LIN {X 0,Y 136.364,Z 311.031,A -85,B 0,C 180,E1 -25968.178,E2 -25968.178} C_VEL
LIN {X 0,Y 134.01,Z 323.173,A -85,B 0,C 180,E1 -25969.777,E2 -25969.777} C_VEL
LIN {X 0,Y 130.975,Z 334.933,A -85,B 0,C 180,E1 -25971.894,E2 -25971.894} C_VEL
LIN {X 0,Y 127.616,Z 346.371,A -85,B 0,C 180,E1 -25974.669,E2 -25974.669} C_VEL
LIN {X 0,Y 124.044,Z 357.11,A -85,B 0,C 180,E1 -25978.099,E2 -25978.099} C_VEL
LIN {X 0,Y 121.088,Z 365.283,A -85,B 0,C 180,E1 -25981.449,E2 -25981.449} C_VEL
LIN {X 0,Y 117.764,Z 374.351,A -85,B 0,C 180,E1 -25986.241,E2 -25986.241} C_VEL
LIN {X 0,Y 115.11,Z 381.715,A -85,B 0,C 180,E1 -25991.301,E2 -25991.301} C_VEL
LIN {X 0,Y 113.643,Z 386.688,A -85,B 0,C 180,E1 -25995.674,E2 -25995.674} C_VEL
LIN {X 0,Y 112.563,Z 391.484,A -85,B 0,C 180,E1 -26001.016,E2 -26001.016} C_VEL
LIN {X 0,Y 112.161,Z 395.114,A -85,B 0,C 180,E1 -26006.404,E2 -26006.404} C_VEL
LIN {X 0,Y 112.247,Z 396.97,A -85,B 0,C 180,E1 -26009.996,E2 -26009.996} C_VEL
LIN {X 0,Y 112.19,Z 398.332,A -85,B 0,C 180,E1 -26013.588,E2 -26013.588} C_VEL
LIN {X 0,Y 112.424,Z 399.289,A -85,B 0,C 180,E1 -26017.178,E2 -26017.178} C_VEL
LIN {X 0,Y 113.828,Z 400.074,A -85,B 0,C 180,E1 -26024.294,E2 -26024.294} C_VEL
LIN {X 0,Y 115.126,Z 399.897,A -85,B 0,C 180,E1 -26027.768,E2 -26027.768} C_VEL
LIN {X 0,Y 118.896,Z 398.375,A -85,B 0,C 180,E1 -26034.438,E2 -26034.438} C_VEL
LIN {X 0,Y 124.439,Z 395.336,A -85,B 0,C 180,E1 -26040.546,E2 -26040.546} C_VEL
LIN {X 0,Y 129.4,Z 391.954,A -85,B 0,C 180,E1 -26044.765,E2 -26044.765} C_VEL
LIN {X 0,Y 134.835,Z 387.585,A -85,B 0,C 180,E1 -26048.712,E2 -26048.712} C_VEL
LIN {X 0,Y 142.27,Z 381.015,A -85,B 0,C 180,E1 -26052.779,E2 -26052.779} C_VEL
LIN {X 0,Y 149.064,Z 373.931,A -85,B 0,C 180,E1 -26055.967,E2 -26055.967} C_VEL
LIN {X 0,Y 156.427,Z 365.2,A -85,B 0,C 180,E1 -26058.806,E2 -26058.806} C_VEL
LIN {X 0,Y 159.478,Z 361.16,A -85,B 0,C 180,E1 -26059.858,E2 -26059.858} C_VEL
LIN {X 0,Y 162.144,Z 357.028,A -85,B 0,C 180,E1 -26061.026,E2 -26061.026} C_VEL
LIN {X 0,Y 165.372,Z 350.19,A -85,B 0,C 180,E1 -26063.269,E2 -26063.269} C_VEL
LIN {X 0,Y 168.431,Z 342.958,A -85,B 0,C 180,E1 -26065.313,E2 -26065.313} C_VEL
LIN {X 0,Y 170.733,Z 338.125,A -85,B 0,C 180,E1 -26066.161,E2 -26066.161} C_VEL
LIN {X 0,Y 176.097,Z 326.328,A -85,B 0,C 180,E1 -26067.398,E2 -26067.398} C_VEL
LIN {X 0,Y 180.609,Z 313.511,A -85,B 0,C 180,E1 -26068.352,E2 -26068.352} C_VEL
LIN {X 0,Y 183.995,Z 300.204,A -85,B 0,C 180,E1 -26069.022,E2 -26069.022} C_VEL
LIN {X 0,Y 186.074,Z 287.077,A -85,B 0,C 180,E1 -26069.451,E2 -26069.451} C_VEL
LIN {X 0,Y 186.09,Z 286.042,A -85,B 0,C 180,E1 -26069.608,E2 -26069.608} C_VEL
LIN {X 0,Y 184.683,Z 281.104,A -85,B 0,C 180,E1 -26072.259,E2 -26072.259} C_VEL
LIN {X 0,Y 183.758,Z 278.277,A -85,B 0,C 180,E1 -26074.485,E2 -26074.485} C_VEL
LIN {X 0,Y 183.075,Z 275.937,A -85,B 0,C 180,E1 -26076.697,E2 -26076.697} C_VEL
LIN {X 0,Y 182.587,Z 274.798,A -85,B 0,C 180,E1 -26078.942,E2 -26078.942} C_VEL
LIN {X 0,Y 182.267,Z 274.378,A -85,B 0,C 180,E1 -26082.032,E2 -26082.032} C_VEL
LIN {X 0,Y 182.898,Z 274.923,A -85,B 0,C 180,E1 -26086.669,E2 -26086.669} C_VEL
LIN {X 0,Y 183.255,Z 275.583,A -85,B 0,C 180,E1 -26087.91,E2 -26087.91} C_VEL
LIN {X 0,Y 184.929,Z 279.204,A -85,B 0,C 180,E1 -26091.984,E2 -26091.984} C_VEL
LIN {X 0,Y 186.439,Z 283.928,A -85,B 0,C 180,E1 -26094.713,E2 -26094.713} C_VEL
LIN {X 0,Y 184.015,Z 299.42,A -85,B 0,C 180,E1 -26095.227,E2 -26095.227} C_VEL
LIN {X 0,Y 180.609,Z 312.589,A -85,B 0,C 180,E1 -26095.931,E2 -26095.931} C_VEL
LIN {X 0,Y 176.382,Z 324.717,A -85,B 0,C 180,E1 -26096.929,E2 -26096.929} C_VEL
LIN {X 0,Y 171.678,Z 335.275,A -85,B 0,C 180,E1 -26098.074,E2 -26098.074} C_VEL
LIN {X 0,Y 165.53,Z 346.46,A -85,B 0,C 180,E1 -26099.672,E2 -26099.672} C_VEL
LIN {X 0,Y 158.442,Z 357.17,A -85,B 0,C 180,E1 -26101.789,E2 -26101.789} C_VEL
LIN {X 0,Y 151.478,Z 365.954,A -85,B 0,C 180,E1 -26104.089,E2 -26104.089} C_VEL
LIN {X 0,Y 145.01,Z 372.979,A -85,B 0,C 180,E1 -26106.549,E2 -26106.549} C_VEL
LIN {X 0,Y 137.992,Z 379.587,A -85,B 0,C 180,E1 -26109.65,E2 -26109.65} C_VEL
LIN {X 0,Y 130.279,Z 385.85,A -85,B 0,C 180,E1 -26113.845,E2 -26113.845} C_VEL
LIN {X 0,Y 122.865,Z 390.935,A -85,B 0,C 180,E1 -26118.918,E2 -26118.918} C_VEL
LIN {X 0,Y 116.03,Z 394.604,A -85,B 0,C 180,E1 -26125.085,E2 -26125.085} C_VEL
LIN {X 0,Y 111.896,Z 396.254,A -85,B 0,C 180,E1 -26130.162,E2 -26130.162} C_VEL
LIN {X 0,Y 108.662,Z 396.997,A -85,B 0,C 180,E1 -26135.596,E2 -26135.596} C_VEL
LIN {X 0,Y 105.831,Z 396.588,A -85,B 0,C 180,E1 -26143.08,E2 -26143.08} C_VEL
LIN {X 0,Y 104.833,Z 395.519,A -85,B 0,C 180,E1 -26147.909,E2 -26147.909} C_VEL
LIN {X 0,Y 104.419,Z 393.352,A -85,B 0,C 180,E1 -26153.866,E2 -26153.866} C_VEL
LIN {X 0,Y 104.975,Z 389.721,A -85,B 0,C 180,E1 -26160.494,E2 -26160.494} C_VEL
LIN {X 0,Y 106.235,Z 385.043,A -85,B 0,C 180,E1 -26166.618,E2 -26166.618} C_VEL
LIN {X 0,Y 108.263,Z 378.481,A -85,B 0,C 180,E1 -26173.021,E2 -26173.021} C_VEL
LIN {X 0,Y 110.851,Z 371.57,A -85,B 0,C 180,E1 -26178.113,E2 -26178.113} C_VEL
LIN {X 0,Y 114.059,Z 363.129,A -85,B 0,C 180,E1 -26182.925,E2 -26182.925} C_VEL
LIN {X 0,Y 117.876,Z 353.263,A -85,B 0,C 180,E1 -26187.218,E2 -26187.218} C_VEL
LIN {X 0,Y 121.724,Z 342.211,A -85,B 0,C 180,E1 -26190.831,E2 -26190.831} C_VEL
LIN {X 0,Y 125.277,Z 330.465,A -85,B 0,C 180,E1 -26193.735,E2 -26193.735} C_VEL
LIN {X 0,Y 128.149,Z 319.202,A -85,B 0,C 180,E1 -26195.808,E2 -26195.808} C_VEL
LIN {X 0,Y 130.747,Z 305.847,A -85,B 0,C 180,E1 -26197.58,E2 -26197.58} C_VEL
LIN {X 0,Y 132.648,Z 292.684,A -85,B 0,C 180,E1 -26198.717,E2 -26198.717} C_VEL
LIN {X 0,Y 136.222,Z 248.968,A -85,B 0,C 180,E1 -26200.99,E2 -26200.99} C_VEL
LIN {X 0,Y 132.344,Z 237.4,A -85,B 0,C 180,E1 -26203.135,E2 -26203.135} C_VEL
LIN {X 0,Y 124.67,Z 222.791,A -85,B 0,C 180,E1 -26207.139,E2 -26207.139} C_VEL
LIN {X 0,Y 118.536,Z 212.859,A -85,B 0,C 180,E1 -26210.752,E2 -26210.752} C_VEL
LIN {X 0,Y 115.586,Z 208.527,A -85,B 0,C 180,E1 -26212.616,E2 -26212.616} C_VEL
LIN {X 0,Y 113.611,Z 205.554,A -85,B 0,C 180,E1 -26213.954,E2 -26213.954} C_VEL
LIN {X 0,Y 111.26,Z 202.05,A -85,B 0,C 180,E1 -26215.65,E2 -26215.65} C_VEL
LIN {X 0,Y 108.737,Z 199.33,A -85,B 0,C 180,E1 -26217.499,E2 -26217.499} C_VEL
LIN {X 0,Y 107.886,Z 197.158,A -85,B 0,C 180,E1 -26218.585,E2 -26218.585} C_VEL
LIN {X 0,Y 107.828,Z 196.58,A -85,B 0,C 180,E1 -26219.804,E2 -26219.804} C_VEL
LIN {X 0,Y 107.715,Z 196.516,A -85,B 0,C 180,E1 -26225.964,E2 -26225.964} C_VEL
LIN {X 0,Y 107.685,Z 196.561,A -85,B 0,C 180,E1 -26230.746,E2 -26230.746} C_VEL
LIN {X 0,Y 107.677,Z 196.518,A -85,B 0,C 180,E1 -26235.891,E2 -26235.891} C_VEL
LIN {X 0,Y 107.687,Z 196.523,A -85,B 0,C 180,E1 -26241.556,E2 -26241.556} C_VEL
LIN {X 0,Y 107.794,Z 196.539,A -85,B 0,C 180,E1 -26248.563,E2 -26248.563} C_VEL
LIN {X 0,Y 107.914,Z 196.522,A -85,B 0,C 180,E1 -26257,E2 -26257} C_VEL
LIN {X 0,Y 108.034,Z 196.506,A -85,B 0,C 180,E1 -26264.919,E2 -26264.919} C_VEL
LIN {X 0,Y 108.254,Z 196.498,A -85,B 0,C 180,E1 -26268.771,E2 -26268.771} C_VEL
LIN {X 0,Y 108.417,Z 196.48,A -85,B 0,C 180,E1 -26276.285,E2 -26276.285} C_VEL
LIN {X 0,Y 108.882,Z 196.374,A -85,B 0,C 180,E1 -26280.002,E2 -26280.002} C_VEL
LIN {X 0,Y 108.295,Z 196.461,A -85,B 0,C 180,E1 -26287.459,E2 -26287.459} C_VEL
LIN {X 0,Y 108.144,Z 196.479,A -85,B 0,C 180,E1 -26292.874,E2 -26292.874} C_VEL
LIN {X 0,Y 107.867,Z 196.515,A -85,B 0,C 180,E1 -26299.014,E2 -26299.014} C_VEL
LIN {X 0,Y 107.826,Z 196.672,A -85,B 0,C 180,E1 -26304.492,E2 -26304.492} C_VEL
LIN {X 0,Y 107.991,Z 197.518,A -85,B 0,C 180,E1 -26305.45,E2 -26305.45} C_VEL
LIN {X 0,Y 109.583,Z 200.432,A -85,B 0,C 180,E1 -26306.935,E2 -26306.935} C_VEL
LIN {X 0,Y 111.163,Z 201.973,A -85,B 0,C 180,E1 -26308.052,E2 -26308.052} C_VEL
LIN {X 0,Y 113.296,Z 205.383,A -85,B 0,C 180,E1 -26309.616,E2 -26309.616} C_VEL
LIN {X 0,Y 114.635,Z 207.06,A -85,B 0,C 180,E1 -26310.503,E2 -26310.503} C_VEL
LIN {X 0,Y 119.745,Z 215.159,A -85,B 0,C 180,E1 -26313.818,E2 -26313.818} C_VEL
LIN {X 0,Y 125.181,Z 224.549,A -85,B 0,C 180,E1 -26316.989,E2 -26316.989} C_VEL
LIN {X 0,Y 128.209,Z 230.807,A -85,B 0,C 180,E1 -26318.671,E2 -26318.671} C_VEL
LIN {X 0,Y 133.626,Z 245.521,A -85,B 0,C 180,E1 -26321.702,E2 -26321.702} C_VEL
LIN {X 0,Y 136.062,Z 253.151,A -85,B 0,C 180,E1 -26323.047,E2 -26323.047} C_VEL
LIN {X 0,Y 132.47,Z 297.001,A -85,B 0,C 180,E1 -26325.357,E2 -26325.357} C_VEL
LIN {X 0,Y 130.339,Z 310.747,A -85,B 0,C 180,E1 -26326.564,E2 -26326.564} C_VEL
LIN {X 0,Y 127.891,Z 322.942,A -85,B 0,C 180,E1 -26328.214,E2 -26328.214} C_VEL
LIN {X 0,Y 124.498,Z 335.522,A -85,B 0,C 180,E1 -26330.571,E2 -26330.571} C_VEL
LIN {X 0,Y 120.993,Z 346.834,A -85,B 0,C 180,E1 -26333.457,E2 -26333.457} C_VEL
LIN {X 0,Y 117.286,Z 357.395,A -85,B 0,C 180,E1 -26337.028,E2 -26337.028} C_VEL
LIN {X 0,Y 114.255,Z 365.435,A -85,B 0,C 180,E1 -26340.518,E2 -26340.518} C_VEL
LIN {X 0,Y 110.755,Z 374.55,A -85,B 0,C 180,E1 -26345.637,E2 -26345.637} C_VEL
LIN {X 0,Y 107.985,Z 381.855,A -85,B 0,C 180,E1 -26351.006,E2 -26351.006} C_VEL
LIN {X 0,Y 106.273,Z 387.67,A -85,B 0,C 180,E1 -26356.613,E2 -26356.613} C_VEL
LIN {X 0,Y 105.316,Z 392.2,A -85,B 0,C 180,E1 -26362.326,E2 -26362.326} C_VEL
LIN {X 0,Y 105.089,Z 394.568,A -85,B 0,C 180,E1 -26366.161,E2 -26366.161} C_VEL
LIN {X 0,Y 105.169,Z 396.493,A -85,B 0,C 180,E1 -26369.996,E2 -26369.996} C_VEL
LIN {X 0,Y 105.108,Z 397.968,A -85,B 0,C 180,E1 -26373.83,E2 -26373.83} C_VEL
LIN {X 0,Y 105.368,Z 399.005,A -85,B 0,C 180,E1 -26377.662,E2 -26377.662} C_VEL
LIN {X 0,Y 106.944,Z 399.927,A -85,B 0,C 180,E1 -26385.236,E2 -26385.236} C_VEL
LIN {X 0,Y 110.154,Z 399.374,A -85,B 0,C 180,E1 -26392.503,E2 -26392.503} C_VEL
LIN {X 0,Y 115.22,Z 397.265,A -85,B 0,C 180,E1 -26399.202,E2 -26399.202} C_VEL
LIN {X 0,Y 121.822,Z 393.613,A -85,B 0,C 180,E1 -26405.228,E2 -26405.228} C_VEL
LIN {X 0,Y 127.627,Z 389.555,A -85,B 0,C 180,E1 -26409.56,E2 -26409.56} C_VEL
LIN {X 0,Y 133.755,Z 384.791,A -85,B 0,C 180,E1 -26413.079,E2 -26413.079} C_VEL
LIN {X 0,Y 141.886,Z 377.496,A -85,B 0,C 180,E1 -26416.932,E2 -26416.932} C_VEL
LIN {X 0,Y 148.117,Z 371.086,A -85,B 0,C 180,E1 -26419.387,E2 -26419.387} C_VEL
LIN {X 0,Y 155.894,Z 361.713,A -85,B 0,C 180,E1 -26422.081,E2 -26422.081} C_VEL
LIN {X 0,Y 163.321,Z 351.079,A -85,B 0,C 180,E1 -26424.308,E2 -26424.308} C_VEL
LIN {X 0,Y 169.699,Z 340.099,A -85,B 0,C 180,E1 -26425.918,E2 -26425.918} C_VEL
LIN {X 0,Y 170.733,Z 338.125,A -85,B 0,C 180,E1 -26426.161,E2 -26426.161} C_VEL
LIN {X 0,Y 172.97,Z 333.179,A -85,B 0,C 180,E1 -26426.963,E2 -26426.963} C_VEL
LIN {X 0,Y 175.622,Z 325.109,A -85,B 0,C 180,E1 -26428.674,E2 -26428.674} C_VEL
LIN {X 0,Y 177.866,Z 316.694,A -85,B 0,C 180,E1 -26430.186,E2 -26430.186} C_VEL
LIN {X 0,Y 179.367,Z 311.228,A -85,B 0,C 180,E1 -26430.68,E2 -26430.68} C_VEL
LIN {X 0,Y 182.606,Z 297.924,A -85,B 0,C 180,E1 -26431.236,E2 -26431.236} C_VEL
LIN {X 0,Y 183.837,Z 290.196,A -85,B 0,C 180,E1 -26431.549,E2 -26431.549} C_VEL
LIN {X 0,Y 182.832,Z 286.166,A -85,B 0,C 180,E1 -26434.026,E2 -26434.026} C_VEL
LIN {X 0,Y 181.855,Z 282.714,A -85,B 0,C 180,E1 -26437.264,E2 -26437.264} C_VEL
LIN {X 0,Y 181.445,Z 281.701,A -85,B 0,C 180,E1 -26439.597,E2 -26439.597} C_VEL
LIN {X 0,Y 181.41,Z 281.461,A -85,B 0,C 180,E1 -26444.264,E2 -26444.264} C_VEL
LIN {X 0,Y 182.006,Z 282.25,A -85,B 0,C 180,E1 -26447.261,E2 -26447.261} C_VEL
LIN {X 0,Y 183.546,Z 285.951,A -85,B 0,C 180,E1 -26451.418,E2 -26451.418} C_VEL
LIN {X 0,Y 184.109,Z 288.316,A -85,B 0,C 180,E1 -26452.72,E2 -26452.72} C_VEL
LIN {X 0,Y 181.696,Z 301.571,A -85,B 0,C 180,E1 -26453.168,E2 -26453.168} C_VEL
LIN {X 0,Y 178.406,Z 313.577,A -85,B 0,C 180,E1 -26453.804,E2 -26453.804} C_VEL
LIN {X 0,Y 173.621,Z 326.545,A -85,B 0,C 180,E1 -26454.856,E2 -26454.856} C_VEL
LIN {X 0,Y 168.174,Z 337.859,A -85,B 0,C 180,E1 -26456.089,E2 -26456.089} C_VEL
LIN {X 0,Y 161.769,Z 348.678,A -85,B 0,C 180,E1 -26457.663,E2 -26457.663} C_VEL
LIN {X 0,Y 154.609,Z 358.712,A -85,B 0,C 180,E1 -26459.664,E2 -26459.664} C_VEL
LIN {X 0,Y 147.654,Z 366.91,A -85,B 0,C 180,E1 -26461.829,E2 -26461.829} C_VEL
LIN {X 0,Y 139.77,Z 374.876,A -85,B 0,C 180,E1 -26464.696,E2 -26464.696} C_VEL
LIN {X 0,Y 131.62,Z 381.86,A -85,B 0,C 180,E1 -26468.216,E2 -26468.216} C_VEL
LIN {X 0,Y 125.487,Z 386.383,A -85,B 0,C 180,E1 -26471.47,E2 -26471.47} C_VEL
LIN {X 0,Y 117.415,Z 391.414,A -85,B 0,C 180,E1 -26476.74,E2 -26476.74} C_VEL
LIN {X 0,Y 110.769,Z 394.663,A -85,B 0,C 180,E1 -26482.374,E2 -26482.374} C_VEL
LIN {X 0,Y 104.866,Z 396.715,A -85,B 0,C 180,E1 -26489.406,E2 -26489.406} C_VEL
LIN {X 0,Y 101.996,Z 397.143,A -85,B 0,C 180,E1 -26494.232,E2 -26494.232} C_VEL
LIN {X 0,Y 99.83,Z 396.974,A -85,B 0,C 180,E1 -26499.314,E2 -26499.314} C_VEL
LIN {X 0,Y 98.047,Z 395.858,A -85,B 0,C 180,E1 -26505.788,E2 -26505.788} C_VEL
LIN {X 0,Y 97.334,Z 393.636,A -85,B 0,C 180,E1 -26512.582,E2 -26512.582} C_VEL
LIN {X 0,Y 97.743,Z 390.021,A -85,B 0,C 180,E1 -26519.786,E2 -26519.786} C_VEL
LIN {X 0,Y 98.644,Z 386.73,A -85,B 0,C 180,E1 -26524.698,E2 -26524.698} C_VEL
LIN {X 0,Y 100.166,Z 381.698,A -85,B 0,C 180,E1 -26530.537,E2 -26530.537} C_VEL
LIN {X 0,Y 102.434,Z 375.417,A -85,B 0,C 180,E1 -26536.176,E2 -26536.176} C_VEL
LIN {X 0,Y 105.445,Z 367.905,A -85,B 0,C 180,E1 -26541.379,E2 -26541.379} C_VEL
LIN {X 0,Y 109.234,Z 358.584,A -85,B 0,C 180,E1 -26546.315,E2 -26546.315} C_VEL
LIN {X 0,Y 113.17,Z 348.266,A -85,B 0,C 180,E1 -26550.448,E2 -26550.448} C_VEL
LIN {X 0,Y 117.139,Z 336.881,A -85,B 0,C 180,E1 -26553.832,E2 -26553.832} C_VEL
LIN {X 0,Y 120.48,Z 325.56,A -85,B 0,C 180,E1 -26556.374,E2 -26556.374} C_VEL
LIN {X 0,Y 123.345,Z 313.358,A -85,B 0,C 180,E1 -26558.399,E2 -26558.399} C_VEL
LIN {X 0,Y 125.893,Z 299.378,A -85,B 0,C 180,E1 -26559.963,E2 -26559.963} C_VEL
LIN {X 0,Y 127.481,Z 285.745,A -85,B 0,C 180,E1 -26560.887,E2 -26560.887} C_VEL
LIN {X 0,Y 130.367,Z 250.585,A -85,B 0,C 180,E1 -26562.745,E2 -26562.745} C_VEL
LIN {X 0,Y 127.215,Z 241.064,A -85,B 0,C 180,E1 -26564.606,E2 -26564.606} C_VEL
LIN {X 0,Y 120.126,Z 227.179,A -85,B 0,C 180,E1 -26568.658,E2 -26568.658} C_VEL
LIN {X 0,Y 112.976,Z 215.35,A -85,B 0,C 180,E1 -26573.258,E2 -26573.258} C_VEL
LIN {X 0,Y 107.405,Z 207.315,A -85,B 0,C 180,E1 -26577.398,E2 -26577.398} C_VEL
LIN {X 0,Y 105.019,Z 204.269,A -85,B 0,C 180,E1 -26579.38,E2 -26579.38} C_VEL
LIN {X 0,Y 104.123,Z 202.586,A -85,B 0,C 180,E1 -26580.229,E2 -26580.229} C_VEL
LIN {X 0,Y 101.914,Z 200.528,A -85,B 0,C 180,E1 -26582.126,E2 -26582.126} C_VEL
LIN {X 0,Y 100.774,Z 198.106,A -85,B 0,C 180,E1 -26583.646,E2 -26583.646} C_VEL
LIN {X 0,Y 100.667,Z 197.442,A -85,B 0,C 180,E1 -26585.172,E2 -26585.172} C_VEL
LIN {X 0,Y 100.643,Z 197.42,A -85,B 0,C 180,E1 -26589.816,E2 -26589.816} C_VEL
LIN {X 0,Y 100.648,Z 197.392,A -85,B 0,C 180,E1 -26595.714,E2 -26595.714} C_VEL
LIN {X 0,Y 100.625,Z 197.394,A -85,B 0,C 180,E1 -26601.056,E2 -26601.056} C_VEL
LIN {X 0,Y 100.691,Z 197.432,A -85,B 0,C 180,E1 -26606.891,E2 -26606.891} C_VEL
LIN {X 0,Y 100.791,Z 197.413,A -85,B 0,C 180,E1 -26615.27,E2 -26615.27} C_VEL
LIN {X 0,Y 100.819,Z 197.419,A -85,B 0,C 180,E1 -26619.604,E2 -26619.604} C_VEL
LIN {X 0,Y 101.104,Z 197.376,A -85,B 0,C 180,E1 -26626.713,E2 -26626.713} C_VEL
LIN {X 0,Y 101.236,Z 197.354,A -85,B 0,C 180,E1 -26632.021,E2 -26632.021} C_VEL
LIN {X 0,Y 101.814,Z 197.251,A -85,B 0,C 180,E1 -26640.002,E2 -26640.002} C_VEL
LIN {X 0,Y 101.232,Z 197.345,A -85,B 0,C 180,E1 -26647.983,E2 -26647.983} C_VEL
LIN {X 0,Y 101.057,Z 197.355,A -85,B 0,C 180,E1 -26653.172,E2 -26653.172} C_VEL
LIN {X 0,Y 100.846,Z 197.647,A -85,B 0,C 180,E1 -26659.598,E2 -26659.598} C_VEL
LIN {X 0,Y 101.057,Z 198.693,A -85,B 0,C 180,E1 -26660.616,E2 -26660.616} C_VEL
LIN {X 0,Y 102.615,Z 201.345,A -85,B 0,C 180,E1 -26662.263,E2 -26662.263} C_VEL
LIN {X 0,Y 104.417,Z 202.965,A -85,B 0,C 180,E1 -26663.82,E2 -26663.82} C_VEL
LIN {X 0,Y 106.359,Z 206.215,A -85,B 0,C 180,E1 -26665.569,E2 -26665.569} C_VEL
LIN {X 0,Y 107.854,Z 207.998,A -85,B 0,C 180,E1 -26666.747,E2 -26666.747} C_VEL
LIN {X 0,Y 110.495,Z 211.755,A -85,B 0,C 180,E1 -26668.753,E2 -26668.753} C_VEL
LIN {X 0,Y 115.819,Z 220.467,A -85,B 0,C 180,E1 -26672.475,E2 -26672.475} C_VEL
LIN {X 0,Y 120.665,Z 229.07,A -85,B 0,C 180,E1 -26675.528,E2 -26675.528} C_VEL
LIN {X 0,Y 123.53,Z 235.191,A -85,B 0,C 180,E1 -26677.266,E2 -26677.266} C_VEL
LIN {X 0,Y 128.851,Z 250.363,A -85,B 0,C 180,E1 -26680.499,E2 -26680.499} C_VEL
LIN {X 0,Y 130.228,Z 254.712,A -85,B 0,C 180,E1 -26681.305,E2 -26681.305} C_VEL
LIN {X 0,Y 126.627,Z 296.718,A -85,B 0,C 180,E1 -26683.574,E2 -26683.574} C_VEL
LIN {X 0,Y 124.551,Z 309.644,A -85,B 0,C 180,E1 -26684.711,E2 -26684.711} C_VEL
LIN {X 0,Y 122.12,Z 321.52,A -85,B 0,C 180,E1 -26686.318,E2 -26686.318} C_VEL
LIN {X 0,Y 119.059,Z 332.845,A -85,B 0,C 180,E1 -26688.384,E2 -26688.384} C_VEL
LIN {X 0,Y 115.342,Z 344.634,A -85,B 0,C 180,E1 -26691.347,E2 -26691.347} C_VEL
LIN {X 0,Y 111.507,Z 355.231,A -85,B 0,C 180,E1 -26694.888,E2 -26694.888} C_VEL
LIN {X 0,Y 108.042,Z 363.889,A -85,B 0,C 180,E1 -26698.638,E2 -26698.638} C_VEL
LIN {X 0,Y 104.836,Z 371.89,A -85,B 0,C 180,E1 -26703.091,E2 -26703.091} C_VEL
LIN {X 0,Y 101.688,Z 379.657,A -85,B 0,C 180,E1 -26708.721,E2 -26708.721} C_VEL
LIN {X 0,Y 99.373,Z 386.808,A -85,B 0,C 180,E1 -26715.664,E2 -26715.664} C_VEL
LIN {X 0,Y 98.281,Z 391.513,A -85,B 0,C 180,E1 -26721.773,E2 -26721.773} C_VEL
LIN {X 0,Y 97.986,Z 395.062,A -85,B 0,C 180,E1 -26727.941,E2 -26727.941} C_VEL
LIN {X 0,Y 98.077,Z 396.001,A -85,B 0,C 180,E1 -26729.996,E2 -26729.996} C_VEL
LIN {X 0,Y 98.049,Z 397.551,A -85,B 0,C 180,E1 -26734.106,E2 -26734.106} C_VEL
LIN {X 0,Y 98.325,Z 398.701,A -85,B 0,C 180,E1 -26738.214,E2 -26738.214} C_VEL
LIN {X 0,Y 100.1,Z 399.78,A -85,B 0,C 180,E1 -26746.306,E2 -26746.306} C_VEL
LIN {X 0,Y 103.606,Z 399.379,A -85,B 0,C 180,E1 -26754.012,E2 -26754.012} C_VEL
LIN {X 0,Y 109.089,Z 397.487,A -85,B 0,C 180,E1 -26761.019,E2 -26761.019} C_VEL
LIN {X 0,Y 116.092,Z 393.991,A -85,B 0,C 180,E1 -26767.251,E2 -26767.251} C_VEL
LIN {X 0,Y 121.863,Z 390.377,A -85,B 0,C 180,E1 -26771.431,E2 -26771.431} C_VEL
LIN {X 0,Y 128.71,Z 385.565,A -85,B 0,C 180,E1 -26775.217,E2 -26775.217} C_VEL
LIN {X 0,Y 137.192,Z 378.554,A -85,B 0,C 180,E1 -26779.073,E2 -26779.073} C_VEL
LIN {X 0,Y 144.984,Z 370.969,A -85,B 0,C 180,E1 -26781.966,E2 -26781.966} C_VEL
LIN {X 0,Y 153.104,Z 361.599,A -85,B 0,C 180,E1 -26784.56,E2 -26784.56} C_VEL
LIN {X 0,Y 160.092,Z 352.085,A -85,B 0,C 180,E1 -26786.515,E2 -26786.515} C_VEL
LIN {X 0,Y 166.667,Z 341.487,A -85,B 0,C 180,E1 -26788.057,E2 -26788.057} C_VEL
LIN {X 0,Y 172.591,Z 329.645,A -85,B 0,C 180,E1 -26789.335,E2 -26789.335} C_VEL
LIN {X 0,Y 177.488,Z 317.232,A -85,B 0,C 180,E1 -26790.297,E2 -26790.297} C_VEL
LIN {X 0,Y 179.367,Z 311.228,A -85,B 0,C 180,E1 -26790.68,E2 -26790.68} C_VEL
LIN {X 0,Y 180.694,Z 305.957,A -85,B 0,C 180,E1 -26791.095,E2 -26791.095} C_VEL
LIN {X 0,Y 181.439,Z 300.97,A -85,B 0,C 180,E1 -26791.859,E2 -26791.859} C_VEL
LIN {X 0,Y 181.708,Z 296.632,A -85,B 0,C 180,E1 -26792.923,E2 -26792.923} C_VEL
LIN {X 0,Y 181.57,Z 293.696,A -85,B 0,C 180,E1 -26794.114,E2 -26794.114} C_VEL
LIN {X 0,Y 181.523,Z 293.372,A -85,B 0,C 180,E1 -26794.303,E2 -26794.303} C_VEL
LIN {X 0,Y 180.725,Z 289.644,A -85,B 0,C 180,E1 -26797.59,E2 -26797.59} C_VEL
LIN {X 0,Y 180.365,Z 288.671,A -85,B 0,C 180,E1 -26799.929,E2 -26799.929} C_VEL
LIN {X 0,Y 180.363,Z 288.482,A -85,B 0,C 180,E1 -26804.17,E2 -26804.17} C_VEL
LIN {X 0,Y 180.84,Z 289.17,A -85,B 0,C 180,E1 -26806.846,E2 -26806.846} C_VEL
LIN {X 0,Y 182.003,Z 292.397,A -85,B 0,C 180,E1 -26810.59,E2 -26810.59} C_VEL
LIN {X 0,Y 180.306,Z 301.139,A -85,B 0,C 180,E1 -26810.954,E2 -26810.954} C_VEL
LIN {X 0,Y 176.611,Z 314.215,A -85,B 0,C 180,E1 -26811.6,E2 -26811.6} C_VEL
LIN {X 0,Y 171.863,Z 326.591,A -85,B 0,C 180,E1 -26812.559,E2 -26812.559} C_VEL
LIN {X 0,Y 166.139,Z 338.122,A -85,B 0,C 180,E1 -26813.739,E2 -26813.739} C_VEL
LIN {X 0,Y 159.814,Z 348.502,A -85,B 0,C 180,E1 -26815.162,E2 -26815.162} C_VEL
LIN {X 0,Y 152.786,Z 358.147,A -85,B 0,C 180,E1 -26816.971,E2 -26816.971} C_VEL
LIN {X 0,Y 144.672,Z 367.339,A -85,B 0,C 180,E1 -26819.266,E2 -26819.266} C_VEL
LIN {X 0,Y 137.101,Z 374.638,A -85,B 0,C 180,E1 -26821.805,E2 -26821.805} C_VEL
LIN {X 0,Y 128.761,Z 381.468,A -85,B 0,C 180,E1 -26825.097,E2 -26825.097} C_VEL
LIN {X 0,Y 120.927,Z 386.935,A -85,B 0,C 180,E1 -26828.913,E2 -26828.913} C_VEL
LIN {X 0,Y 115.107,Z 390.371,A -85,B 0,C 180,E1 -26832.361,E2 -26832.361} C_VEL
LIN {X 0,Y 109.739,Z 393.092,A -85,B 0,C 180,E1 -26836.144,E2 -26836.144} C_VEL
LIN {X 0,Y 104.883,Z 395.095,A -85,B 0,C 180,E1 -26840.277,E2 -26840.277} C_VEL
LIN {X 0,Y 100.653,Z 396.442,A -85,B 0,C 180,E1 -26844.821,E2 -26844.821} C_VEL
LIN {X 0,Y 96.519,Z 397.228,A -85,B 0,C 180,E1 -26850.642,E2 -26850.642} C_VEL
LIN {X 0,Y 93.409,Z 397.117,A -85,B 0,C 180,E1 -26857.005,E2 -26857.005} C_VEL
LIN {X 0,Y 91.304,Z 396.042,A -85,B 0,C 180,E1 -26863.847,E2 -26863.847} C_VEL
LIN {X 0,Y 90.266,Z 393.745,A -85,B 0,C 180,E1 -26871.481,E2 -26871.481} C_VEL
LIN {X 0,Y 90.498,Z 390.474,A -85,B 0,C 180,E1 -26878.673,E2 -26878.673} C_VEL
LIN {X 0,Y 91.491,Z 386.774,A -85,B 0,C 180,E1 -26884.694,E2 -26884.694} C_VEL
LIN {X 0,Y 93.204,Z 381.405,A -85,B 0,C 180,E1 -26891.314,E2 -26891.314} C_VEL
LIN {X 0,Y 95.597,Z 375.115,A -85,B 0,C 180,E1 -26897.263,E2 -26897.263} C_VEL
LIN {X 0,Y 99.087,Z 366.874,A -85,B 0,C 180,E1 -26903.193,E2 -26903.193} C_VEL
LIN {X 0,Y 102.912,Z 357.96,A -85,B 0,C 180,E1 -26908.047,E2 -26908.047} C_VEL
LIN {X 0,Y 106.618,Z 348.73,A -85,B 0,C 180,E1 -26911.893,E2 -26911.893} C_VEL
LIN {X 0,Y 110.81,Z 337.269,A -85,B 0,C 180,E1 -26915.463,E2 -26915.463} C_VEL
LIN {X 0,Y 114.148,Z 326.606,A -85,B 0,C 180,E1 -26917.966,E2 -26917.966} C_VEL
LIN {X 0,Y 117.271,Z 314.197,A -85,B 0,C 180,E1 -26920.143,E2 -26920.143} C_VEL
LIN {X 0,Y 119.828,Z 300.782,A -85,B 0,C 180,E1 -26921.736,E2 -26921.736} C_VEL
LIN {X 0,Y 121.525,Z 288.176,A -85,B 0,C 180,E1 -26922.657,E2 -26922.657} C_VEL
LIN {X 0,Y 124.569,Z 252.247,A -85,B 0,C 180,E1 -26924.627,E2 -26924.627} C_VEL
LIN {X 0,Y 122.216,Z 244.873,A -85,B 0,C 180,E1 -26926.171,E2 -26926.171} C_VEL
LIN {X 0,Y 115.71,Z 231.709,A -85,B 0,C 180,E1 -26930.222,E2 -26930.222} C_VEL
LIN {X 0,Y 109.001,Z 220.387,A -85,B 0,C 180,E1 -26934.909,E2 -26934.909} C_VEL
LIN {X 0,Y 103.911,Z 212.805,A -85,B 0,C 180,E1 -26939.052,E2 -26939.052} C_VEL
LIN {X 0,Y 101.394,Z 209.255,A -85,B 0,C 180,E1 -26941.336,E2 -26941.336} C_VEL
LIN {X 0,Y 98.327,Z 205.356,A -85,B 0,C 180,E1 -26944.348,E2 -26944.348} C_VEL
LIN {X 0,Y 97.317,Z 203.694,A -85,B 0,C 180,E1 -26945.496,E2 -26945.496} C_VEL
LIN {X 0,Y 94.829,Z 201.514,A -85,B 0,C 180,E1 -26948.269,E2 -26948.269} C_VEL
LIN {X 0,Y 93.666,Z 198.881,A -85,B 0,C 180,E1 -26950.41,E2 -26950.41} C_VEL
LIN {X 0,Y 93.537,Z 198.355,A -85,B 0,C 180,E1 -26952.554,E2 -26952.554} C_VEL
LIN {X 0,Y 93.535,Z 198.262,A -85,B 0,C 180,E1 -26958.715,E2 -26958.715} C_VEL
LIN {X 0,Y 93.589,Z 198.326,A -85,B 0,C 180,E1 -26965.701,E2 -26965.701} C_VEL
LIN {X 0,Y 93.672,Z 198.307,A -85,B 0,C 180,E1 -26974.21,E2 -26974.21} C_VEL
LIN {X 0,Y 93.695,Z 198.294,A -85,B 0,C 180,E1 -26977.975,E2 -26977.975} C_VEL
LIN {X 0,Y 94.024,Z 198.255,A -85,B 0,C 180,E1 -26986.353,E2 -26986.353} C_VEL
LIN {X 0,Y 94.171,Z 198.234,A -85,B 0,C 180,E1 -26991.418,E2 -26991.418} C_VEL
LIN {X 0,Y 94.746,Z 198.128,A -85,B 0,C 180,E1 -27000.002,E2 -27000.002} C_VEL
LIN {X 0,Y 94.163,Z 198.232,A -85,B 0,C 180,E1 -27008.587,E2 -27008.587} C_VEL
LIN {X 0,Y 94.046,Z 198.533,A -85,B 0,C 180,E1 -27013.259,E2 -27013.259} C_VEL
LIN {X 0,Y 94.275,Z 199.852,A -85,B 0,C 180,E1 -27014.573,E2 -27014.573} C_VEL
LIN {X 0,Y 95.918,Z 202.489,A -85,B 0,C 180,E1 -27016.77,E2 -27016.77} C_VEL
LIN {X 0,Y 97.671,Z 203.923,A -85,B 0,C 180,E1 -27018.623,E2 -27018.623} C_VEL
LIN {X 0,Y 99.649,Z 207.242,A -85,B 0,C 180,E1 -27020.78,E2 -27020.78} C_VEL
LIN {X 0,Y 101.42,Z 209.192,A -85,B 0,C 180,E1 -27022.44,E2 -27022.44} C_VEL
LIN {X 0,Y 103.802,Z 212.673,A -85,B 0,C 180,E1 -27024.635,E2 -27024.635} C_VEL
LIN {X 0,Y 109.101,Z 220.772,A -85,B 0,C 180,E1 -27028.958,E2 -27028.958} C_VEL
LIN {X 0,Y 115.212,Z 231.613,A -85,B 0,C 180,E1 -27033.301,E2 -27033.301} C_VEL
LIN {X 0,Y 118.499,Z 238.477,A -85,B 0,C 180,E1 -27035.46,E2 -27035.46} C_VEL
LIN {X 0,Y 123.596,Z 253.579,A -85,B 0,C 180,E1 -27038.894,E2 -27038.894} C_VEL
LIN {X 0,Y 124.495,Z 256.636,A -85,B 0,C 180,E1 -27039.487,E2 -27039.487} C_VEL
LIN {X 0,Y 120.854,Z 296.514,A -85,B 0,C 180,E1 -27041.673,E2 -27041.673} C_VEL
LIN {X 0,Y 118.652,Z 309.698,A -85,B 0,C 180,E1 -27042.858,E2 -27042.858} C_VEL
LIN {X 0,Y 115.976,Z 322.083,A -85,B 0,C 180,E1 -27044.595,E2 -27044.595} C_VEL
LIN {X 0,Y 112.792,Z 333.249,A -85,B 0,C 180,E1 -27046.729,E2 -27046.729} C_VEL
LIN {X 0,Y 108.901,Z 344.919,A -85,B 0,C 180,E1 -27049.803,E2 -27049.803} C_VEL
LIN {X 0,Y 104.763,Z 355.731,A -85,B 0,C 180,E1 -27053.614,E2 -27053.614} C_VEL
LIN {X 0,Y 101.275,Z 364.058,A -85,B 0,C 180,E1 -27057.461,E2 -27057.461} C_VEL
LIN {X 0,Y 97.898,Z 372.005,A -85,B 0,C 180,E1 -27062.18,E2 -27062.18} C_VEL
LIN {X 0,Y 94.6,Z 379.717,A -85,B 0,C 180,E1 -27068.19,E2 -27068.19} C_VEL
LIN {X 0,Y 92.49,Z 385.92,A -85,B 0,C 180,E1 -27074.572,E2 -27074.572} C_VEL
LIN {X 0,Y 91.27,Z 390.794,A -85,B 0,C 180,E1 -27081.136,E2 -27081.136} C_VEL
LIN {X 0,Y 90.901,Z 394.496,A -85,B 0,C 180,E1 -27087.78,E2 -27087.78} C_VEL
LIN {X 0,Y 90.996,Z 395.507,A -85,B 0,C 180,E1 -27089.995,E2 -27089.995} C_VEL
LIN {X 0,Y 90.98,Z 397.12,A -85,B 0,C 180,E1 -27094.426,E2 -27094.426} C_VEL
LIN {X 0,Y 92.069,Z 399.173,A -85,B 0,C 180,E1 -27103.233,E2 -27103.233} C_VEL
LIN {X 0,Y 93.303,Z 399.629,A -85,B 0,C 180,E1 -27107.531,E2 -27107.531} C_VEL
LIN {X 0,Y 97.144,Z 399.378,A -85,B 0,C 180,E1 -27115.721,E2 -27115.721} C_VEL
LIN {X 0,Y 103.081,Z 397.673,A -85,B 0,C 180,E1 -27123.049,E2 -27123.049} C_VEL
LIN {X 0,Y 106.638,Z 396.253,A -85,B 0,C 180,E1 -27126.375,E2 -27126.375} C_VEL
LIN {X 0,Y 112.54,Z 393.357,A -85,B 0,C 180,E1 -27130.968,E2 -27130.968} C_VEL
LIN {X 0,Y 119.058,Z 389.499,A -85,B 0,C 180,E1 -27135.096,E2 -27135.096} C_VEL
LIN {X 0,Y 126.325,Z 384.566,A -85,B 0,C 180,E1 -27138.676,E2 -27138.676} C_VEL
LIN {X 0,Y 135.292,Z 377.313,A -85,B 0,C 180,E1 -27142.384,E2 -27142.384} C_VEL
LIN {X 0,Y 143.521,Z 369.502,A -85,B 0,C 180,E1 -27145.1,E2 -27145.1} C_VEL
LIN {X 0,Y 152.064,Z 359.884,A -85,B 0,C 180,E1 -27147.502,E2 -27147.502} C_VEL
LIN {X 0,Y 159.364,Z 349.931,A -85,B 0,C 180,E1 -27149.305,E2 -27149.305} C_VEL
LIN {X 0,Y 166.14,Z 338.82,A -85,B 0,C 180,E1 -27150.74,E2 -27150.74} C_VEL
LIN {X 0,Y 171.478,Z 328.059,A -85,B 0,C 180,E1 -27151.778,E2 -27151.778} C_VEL
LIN {X 0,Y 176.04,Z 316.576,A -85,B 0,C 180,E1 -27152.583,E2 -27152.583} C_VEL
LIN {X 0,Y 179.731,Z 304.026,A -85,B 0,C 180,E1 -27153.211,E2 -27153.211} C_VEL
LIN {X 0,Y 181.741,Z 294.459,A -85,B 0,C 180,E1 -27153.574,E2 -27153.574} C_VEL
LIN {X 0,Y 181.523,Z 293.372,A -85,B 0,C 180,E1 -27154.303,E2 -27154.303} C_VEL
LIN {X 0,Y 181.168,Z 292.097,A -85,B 0,C 180,E1 -27155.46,E2 -27155.46} C_VEL
LIN {X 0,Y 180.509,Z 291.677,A -85,B 0,C 180,E1 -27157.311,E2 -27157.311} C_VEL
LIN {X 0,Y 179.869,Z 292.441,A -85,B 0,C 180,E1 -27159.185,E2 -27159.185} C_VEL
LIN {X 0,Y 179.11,Z 295.072,A -85,B 0,C 180,E1 -27163.081,E2 -27163.081} C_VEL
LIN {X 0,Y 179.164,Z 295.519,A -85,B 0,C 180,E1 -27164.402,E2 -27164.402} C_VEL
LIN {X 0,Y 179.486,Z 296.168,A -85,B 0,C 180,E1 -27166.578,E2 -27166.578} C_VEL
LIN {X 0,Y 179.875,Z 297.901,A -85,B 0,C 180,E1 -27168.612,E2 -27168.612} C_VEL
LIN {X 0,Y 176.49,Z 310.901,A -85,B 0,C 180,E1 -27169.139,E2 -27169.139} C_VEL
LIN {X 0,Y 172.111,Z 322.913,A -85,B 0,C 180,E1 -27169.914,E2 -27169.914} C_VEL
LIN {X 0,Y 166.097,Z 335.537,A -85,B 0,C 180,E1 -27171.005,E2 -27171.005} C_VEL
LIN {X 0,Y 159.251,Z 346.845,A -85,B 0,C 180,E1 -27172.391,E2 -27172.391} C_VEL
LIN {X 0,Y 152.294,Z 356.31,A -85,B 0,C 180,E1 -27173.959,E2 -27173.959} C_VEL
LIN {X 0,Y 144.426,Z 365.318,A -85,B 0,C 180,E1 -27175.945,E2 -27175.945} C_VEL
LIN {X 0,Y 137.114,Z 372.426,A -85,B 0,C 180,E1 -27178.067,E2 -27178.067} C_VEL
LIN {X 0,Y 128.92,Z 379.238,A -85,B 0,C 180,E1 -27180.856,E2 -27180.856} C_VEL
LIN {X 0,Y 119.848,Z 385.512,A -85,B 0,C 180,E1 -27184.573,E2 -27184.573} C_VEL
LIN {X 0,Y 110.468,Z 390.824,A -85,B 0,C 180,E1 -27189.598,E2 -27189.598} C_VEL
LIN {X 0,Y 102.066,Z 394.514,A -85,B 0,C 180,E1 -27195.439,E2 -27195.439} C_VEL
LIN {X 0,Y 95.499,Z 396.532,A -85,B 0,C 180,E1 -27201.588,E2 -27201.588} C_VEL
LIN {X 0,Y 89.316,Z 397.413,A -85,B 0,C 180,E1 -27210.065,E2 -27210.065} C_VEL
LIN {X 0,Y 86.587,Z 397.104,A -85,B 0,C 180,E1 -27215.75,E2 -27215.75} C_VEL
LIN {X 0,Y 84.646,Z 396.206,A -85,B 0,C 180,E1 -27221.656,E2 -27221.656} C_VEL
LIN {X 0,Y 83.3,Z 394.118,A -85,B 0,C 180,E1 -27229.401,E2 -27229.401} C_VEL
LIN {X 0,Y 83.292,Z 390.801,A -85,B 0,C 180,E1 -27237.537,E2 -27237.537} C_VEL
LIN {X 0,Y 84.606,Z 385.848,A -85,B 0,C 180,E1 -27246.022,E2 -27246.022} C_VEL
LIN {X 0,Y 86.623,Z 380.168,A -85,B 0,C 180,E1 -27253.197,E2 -27253.197} C_VEL
LIN {X 0,Y 89.499,Z 373.245,A -85,B 0,C 180,E1 -27259.828,E2 -27259.828} C_VEL
LIN {X 0,Y 93.105,Z 365.151,A -85,B 0,C 180,E1 -27265.676,E2 -27265.676} C_VEL
LIN {X 0,Y 97.701,Z 354.998,A -85,B 0,C 180,E1 -27271.066,E2 -27271.066} C_VEL
LIN {X 0,Y 101.744,Z 345.21,A -85,B 0,C 180,E1 -27274.957,E2 -27274.957} C_VEL
LIN {X 0,Y 105.596,Z 334.819,A -85,B 0,C 180,E1 -27278.065,E2 -27278.065} C_VEL
LIN {X 0,Y 109.332,Z 322.772,A -85,B 0,C 180,E1 -27280.73,E2 -27280.73} C_VEL
LIN {X 0,Y 112.552,Z 309.443,A -85,B 0,C 180,E1 -27282.857,E2 -27282.857} C_VEL
LIN {X 0,Y 114.981,Z 295.815,A -85,B 0,C 180,E1 -27284.233,E2 -27284.233} C_VEL
LIN {X 0,Y 117.482,Z 271.81,A -85,B 0,C 180,E1 -27285.635,E2 -27285.635} C_VEL
LIN {X 0,Y 118.963,Z 253.945,A -85,B 0,C 180,E1 -27286.671,E2 -27286.671} C_VEL
LIN {X 0,Y 117.238,Z 248.436,A -85,B 0,C 180,E1 -27287.926,E2 -27287.926} C_VEL
LIN {X 0,Y 111.284,Z 236.047,A -85,B 0,C 180,E1 -27291.949,E2 -27291.949} C_VEL
LIN {X 0,Y 105.08,Z 225.287,A -85,B 0,C 180,E1 -27296.727,E2 -27296.727} C_VEL
LIN {X 0,Y 100.52,Z 218.361,A -85,B 0,C 180,E1 -27300.739,E2 -27300.739} C_VEL
LIN {X 0,Y 97.569,Z 214.12,A -85,B 0,C 180,E1 -27303.692,E2 -27303.692} C_VEL
LIN {X 0,Y 95.099,Z 210.557,A -85,B 0,C 180,E1 -27306.479,E2 -27306.479} C_VEL
LIN {X 0,Y 93.807,Z 209.262,A -85,B 0,C 180,E1 -27307.992,E2 -27307.992} C_VEL
LIN {X 0,Y 91.752,Z 206.632,A -85,B 0,C 180,E1 -27310.738,E2 -27310.738} C_VEL
LIN {X 0,Y 90.798,Z 204.922,A -85,B 0,C 180,E1 -27312.212,E2 -27312.212} C_VEL
LIN {X 0,Y 88.181,Z 203.03,A -85,B 0,C 180,E1 -27316.114,E2 -27316.114} C_VEL
LIN {X 0,Y 86.55,Z 199.833,A -85,B 0,C 180,E1 -27320.173,E2 -27320.173} C_VEL
LIN {X 0,Y 86.484,Z 199.226,A -85,B 0,C 180,E1 -27323.46,E2 -27323.46} C_VEL
LIN {X 0,Y 86.475,Z 199.197,A -85,B 0,C 180,E1 -27330.817,E2 -27330.817} C_VEL
LIN {X 0,Y 86.59,Z 199.177,A -85,B 0,C 180,E1 -27336.06,E2 -27336.06} C_VEL
LIN {X 0,Y 86.665,Z 199.186,A -85,B 0,C 180,E1 -27341.074,E2 -27341.074} C_VEL
LIN {X 0,Y 86.937,Z 199.134,A -85,B 0,C 180,E1 -27345.967,E2 -27345.967} C_VEL
LIN {X 0,Y 87.082,Z 199.119,A -85,B 0,C 180,E1 -27350.713,E2 -27350.713} C_VEL
LIN {X 0,Y 87.678,Z 199.005,A -85,B 0,C 180,E1 -27360.002,E2 -27360.002} C_VEL
LIN {X 0,Y 87.272,Z 199.465,A -85,B 0,C 180,E1 -27364.332,E2 -27364.332} C_VEL
LIN {X 0,Y 87.578,Z 200.809,A -85,B 0,C 180,E1 -27366.048,E2 -27366.048} C_VEL
LIN {X 0,Y 89.167,Z 203.309,A -85,B 0,C 180,E1 -27369.072,E2 -27369.072} C_VEL
LIN {X 0,Y 91.362,Z 205.151,A -85,B 0,C 180,E1 -27372.3,E2 -27372.3} C_VEL
LIN {X 0,Y 93.16,Z 208.388,A -85,B 0,C 180,E1 -27374.964,E2 -27374.964} C_VEL
LIN {X 0,Y 95.032,Z 210.405,A -85,B 0,C 180,E1 -27377.209,E2 -27377.209} C_VEL
LIN {X 0,Y 97.339,Z 213.823,A -85,B 0,C 180,E1 -27379.828,E2 -27379.828} C_VEL
LIN {X 0,Y 98.561,Z 215.49,A -85,B 0,C 180,E1 -27381.085,E2 -27381.085} C_VEL
LIN {X 0,Y 101.613,Z 220.096,A -85,B 0,C 180,E1 -27384.06,E2 -27384.06} C_VEL
LIN {X 0,Y 105.506,Z 226.29,A -85,B 0,C 180,E1 -27387.442,E2 -27387.442} C_VEL
LIN {X 0,Y 110.94,Z 236.242,A -85,B 0,C 180,E1 -27391.664,E2 -27391.664} C_VEL
LIN {X 0,Y 113.73,Z 242.257,A -85,B 0,C 180,E1 -27393.666,E2 -27393.666} C_VEL
LIN {X 0,Y 118.478,Z 256.903,A -85,B 0,C 180,E1 -27397.173,E2 -27397.173} C_VEL
LIN {X 0,Y 118.844,Z 258.733,A -85,B 0,C 180,E1 -27397.492,E2 -27397.492} C_VEL
LIN {X 0,Y 115.222,Z 296.279,A -85,B 0,C 180,E1 -27399.578,E2 -27399.578} C_VEL
LIN {X 0,Y 112.987,Z 309.307,A -85,B 0,C 180,E1 -27400.765,E2 -27400.765} C_VEL
LIN {X 0,Y 110.232,Z 321.544,A -85,B 0,C 180,E1 -27402.503,E2 -27402.503} C_VEL
LIN {X 0,Y 106.61,Z 333.616,A -85,B 0,C 180,E1 -27404.869,E2 -27404.869} C_VEL
LIN {X 0,Y 102.558,Z 345.207,A -85,B 0,C 180,E1 -27408.072,E2 -27408.072} C_VEL
LIN {X 0,Y 98.658,Z 354.845,A -85,B 0,C 180,E1 -27411.594,E2 -27411.594} C_VEL
LIN {X 0,Y 94.541,Z 364.222,A -85,B 0,C 180,E1 -27416.11,E2 -27416.11} C_VEL
LIN {X 0,Y 90.382,Z 373.48,A -85,B 0,C 180,E1 -27422.184,E2 -27422.184} C_VEL
LIN {X 0,Y 87.116,Z 380.89,A -85,B 0,C 180,E1 -27428.709,E2 -27428.709} C_VEL
LIN {X 0,Y 85.061,Z 386.827,A -85,B 0,C 180,E1 -27435.644,E2 -27435.644} C_VEL
LIN {X 0,Y 84.031,Z 391.465,A -85,B 0,C 180,E1 -27442.788,E2 -27442.788} C_VEL
LIN {X 0,Y 83.916,Z 394.949,A -85,B 0,C 180,E1 -27449.995,E2 -27449.995} C_VEL
LIN {X 0,Y 83.931,Z 396.673,A -85,B 0,C 180,E1 -27454.798,E2 -27454.798} C_VEL
LIN {X 0,Y 85.174,Z 398.876,A -85,B 0,C 180,E1 -27464.327,E2 -27464.327} C_VEL
LIN {X 0,Y 88.39,Z 399.594,A -85,B 0,C 180,E1 -27473.42,E2 -27473.42} C_VEL
LIN {X 0,Y 93.767,Z 398.794,A -85,B 0,C 180,E1 -27481.64,E2 -27481.64} C_VEL
LIN {X 0,Y 101.001,Z 396.519,A -85,B 0,C 180,E1 -27488.768,E2 -27488.768} C_VEL
LIN {X 0,Y 107.284,Z 393.775,A -85,B 0,C 180,E1 -27493.453,E2 -27493.453} C_VEL
LIN {X 0,Y 114.173,Z 390.103,A -85,B 0,C 180,E1 -27497.612,E2 -27497.612} C_VEL
LIN {X 0,Y 121.796,Z 385.392,A -85,B 0,C 180,E1 -27501.162,E2 -27501.162} C_VEL
LIN {X 0,Y 131.13,Z 378.451,A -85,B 0,C 180,E1 -27504.812,E2 -27504.812} C_VEL
LIN {X 0,Y 139.663,Z 370.935,A -85,B 0,C 180,E1 -27507.438,E2 -27507.438} C_VEL
LIN {X 0,Y 148.446,Z 361.622,A -85,B 0,C 180,E1 -27509.764,E2 -27509.764} C_VEL
LIN {X 0,Y 156.713,Z 351.139,A -85,B 0,C 180,E1 -27511.648,E2 -27511.648} C_VEL
LIN {X 0,Y 163.661,Z 340.388,A -85,B 0,C 180,E1 -27512.999,E2 -27512.999} C_VEL
LIN {X 0,Y 169.908,Z 328.41,A -85,B 0,C 180,E1 -27514.106,E2 -27514.106} C_VEL
LIN {X 0,Y 174.714,Z 316.679,A -85,B 0,C 180,E1 -27514.876,E2 -27514.876} C_VEL
LIN {X 0,Y 178.635,Z 303.625,A -85,B 0,C 180,E1 -27515.47,E2 -27515.47} C_VEL
LIN {X 0,Y 179.696,Z 299.117,A -85,B 0,C 180,E1 -27515.609,E2 -27515.609} C_VEL
LIN {X 0,Y 179.302,Z 296.231,A -85,B 0,C 180,E1 -27518.495,E2 -27518.495} C_VEL
LIN {X 0,Y 179.102,Z 295.587,A -85,B 0,C 180,E1 -27520.341,E2 -27520.341} C_VEL
LIN {X 0,Y 179.164,Z 295.519,A -85,B 0,C 180,E1 -27524.402,E2 -27524.402} C_VEL
LIN {X 0,Y 179.098,Z 296.512,A -85,B 0,C 180,E1 -27525.219,E2 -27525.219} C_VEL
LIN {X 0,Y 178.698,Z 299.111,A -85,B 0,C 180,E1 -27525.967,E2 -27525.967} C_VEL
LIN {X 0,Y 177.914,Z 302.711,A -85,B 0,C 180,E1 -27526.465,E2 -27526.465} C_VEL
LIN {X 0,Y 176.294,Z 308.675,A -85,B 0,C 180,E1 -27526.816,E2 -27526.816} C_VEL
LIN {X 0,Y 174.329,Z 314.627,A -85,B 0,C 180,E1 -27527.019,E2 -27527.019} C_VEL
LIN {X 0,Y 169.669,Z 326.238,A -85,B 0,C 180,E1 -27527.782,E2 -27527.782} C_VEL
LIN {X 0,Y 163.969,Z 337.308,A -85,B 0,C 180,E1 -27528.721,E2 -27528.721} C_VEL
LIN {X 0,Y 156.99,Z 348.252,A -85,B 0,C 180,E1 -27530.003,E2 -27530.003} C_VEL
LIN {X 0,Y 149.167,Z 358.341,A -85,B 0,C 180,E1 -27531.631,E2 -27531.631} C_VEL
LIN {X 0,Y 141.487,Z 366.564,A -85,B 0,C 180,E1 -27533.403,E2 -27533.403} C_VEL
LIN {X 0,Y 132.587,Z 374.548,A -85,B 0,C 180,E1 -27535.812,E2 -27535.812} C_VEL
LIN {X 0,Y 123.088,Z 381.667,A -85,B 0,C 180,E1 -27538.907,E2 -27538.907} C_VEL
LIN {X 0,Y 116.002,Z 386.134,A -85,B 0,C 180,E1 -27541.67,E2 -27541.67} C_VEL
LIN {X 0,Y 106.112,Z 391.319,A -85,B 0,C 180,E1 -27546.587,E2 -27546.587} C_VEL
LIN {X 0,Y 96.982,Z 394.884,A -85,B 0,C 180,E1 -27552.554,E2 -27552.554} C_VEL
LIN {X 0,Y 89.39,Z 396.886,A -85,B 0,C 180,E1 -27559.375,E2 -27559.375} C_VEL
LIN {X 0,Y 85.066,Z 397.474,A -85,B 0,C 180,E1 -27564.673,E2 -27564.673} C_VEL
LIN {X 0,Y 81.137,Z 397.386,A -85,B 0,C 180,E1 -27571.311,E2 -27571.311} C_VEL
LIN {X 0,Y 78.124,Z 396.366,A -85,B 0,C 180,E1 -27579.026,E2 -27579.026} C_VEL
LIN {X 0,Y 76.406,Z 394.332,A -85,B 0,C 180,E1 -27587.376,E2 -27587.376} C_VEL
LIN {X 0,Y 76.119,Z 391.037,A -85,B 0,C 180,E1 -27596.367,E2 -27596.367} C_VEL
LIN {X 0,Y 77.303,Z 386.304,A -85,B 0,C 180,E1 -27605.382,E2 -27605.382} C_VEL
LIN {X 0,Y 79.374,Z 380.663,A -85,B 0,C 180,E1 -27613.282,E2 -27613.282} C_VEL
LIN {X 0,Y 82.818,Z 372.835,A -85,B 0,C 180,E1 -27621.39,E2 -27621.39} C_VEL
LIN {X 0,Y 86.753,Z 364.474,A -85,B 0,C 180,E1 -27627.683,E2 -27627.683} C_VEL
LIN {X 0,Y 91.496,Z 354.604,A -85,B 0,C 180,E1 -27633.116,E2 -27633.116} C_VEL
LIN {X 0,Y 96.04,Z 344.127,A -85,B 0,C 180,E1 -27637.362,E2 -27637.362} C_VEL
LIN {X 0,Y 100.613,Z 331.955,A -85,B 0,C 180,E1 -27640.931,E2 -27640.931} C_VEL
LIN {X 0,Y 104.262,Z 320.336,A -85,B 0,C 180,E1 -27643.402,E2 -27643.402} C_VEL
LIN {X 0,Y 107.333,Z 307.374,A -85,B 0,C 180,E1 -27645.368,E2 -27645.368} C_VEL
LIN {X 0,Y 109.772,Z 293.623,A -85,B 0,C 180,E1 -27646.683,E2 -27646.683} C_VEL
LIN {X 0,Y 113.532,Z 256.6,A -85,B 0,C 180,E1 -27648.767,E2 -27648.767} C_VEL
LIN {X 0,Y 112.898,Z 253.433,A -85,B 0,C 180,E1 -27649.37,E2 -27649.37} C_VEL
LIN {X 0,Y 107.061,Z 240.608,A -85,B 0,C 180,E1 -27653.737,E2 -27653.737} C_VEL
LIN {X 0,Y 101.253,Z 230.256,A -85,B 0,C 180,E1 -27658.621,E2 -27658.621} C_VEL
LIN {X 0,Y 97.131,Z 223.732,A -85,B 0,C 180,E1 -27662.645,E2 -27662.645} C_VEL
LIN {X 0,Y 94.479,Z 219.752,A -85,B 0,C 180,E1 -27665.578,E2 -27665.578} C_VEL
LIN {X 0,Y 91.893,Z 215.962,A -85,B 0,C 180,E1 -27668.835,E2 -27668.835} C_VEL
LIN {X 0,Y 89.501,Z 213.105,A -85,B 0,C 180,E1 -27672.161,E2 -27672.161} C_VEL
LIN {X 0,Y 88.706,Z 211.525,A -85,B 0,C 180,E1 -27673.503,E2 -27673.503} C_VEL
LIN {X 0,Y 86.058,Z 209.238,A -85,B 0,C 180,E1 -27677.924,E2 -27677.924} C_VEL
LIN {X 0,Y 84.45,Z 206.226,A -85,B 0,C 180,E1 -27681.763,E2 -27681.763} C_VEL
LIN {X 0,Y 80.521,Z 202.912,A -85,B 0,C 180,E1 -27696.876,E2 -27696.876} C_VEL
LIN {X 0,Y 80.43,Z 202.263,A -85,B 0,C 180,E1 -27704.805,E2 -27704.805} C_VEL
LIN {X 0,Y 81.209,Z 203.135,A -85,B 0,C 180,E1 -27711.291,E2 -27711.291} C_VEL
LIN {X 0,Y 84.494,Z 205.546,A -85,B 0,C 180,E1 -27721.847,E2 -27721.847} C_VEL
LIN {X 0,Y 85.241,Z 206.383,A -85,B 0,C 180,E1 -27723.546,E2 -27723.546} C_VEL
LIN {X 0,Y 86.791,Z 209.308,A -85,B 0,C 180,E1 -27726.979,E2 -27726.979} C_VEL
LIN {X 0,Y 89.033,Z 211.593,A -85,B 0,C 180,E1 -27730.693,E2 -27730.693} C_VEL
LIN {X 0,Y 91.19,Z 215.104,A -85,B 0,C 180,E1 -27734.01,E2 -27734.01} C_VEL
LIN {X 0,Y 92.452,Z 216.662,A -85,B 0,C 180,E1 -27735.673,E2 -27735.673} C_VEL
LIN {X 0,Y 95.716,Z 221.596,A -85,B 0,C 180,E1 -27739.598,E2 -27739.598} C_VEL
LIN {X 0,Y 98.54,Z 226.05,A -85,B 0,C 180,E1 -27742.592,E2 -27742.592} C_VEL
LIN {X 0,Y 101.762,Z 231.366,A -85,B 0,C 180,E1 -27745.634,E2 -27745.634} C_VEL
LIN {X 0,Y 106.815,Z 241.034,A -85,B 0,C 180,E1 -27749.944,E2 -27749.944} C_VEL
LIN {X 0,Y 109.072,Z 246.173,A -85,B 0,C 180,E1 -27751.752,E2 -27751.752} C_VEL
LIN {X 0,Y 113.304,Z 259.672,A -85,B 0,C 180,E1 -27755.197,E2 -27755.197} C_VEL
LIN {X 0,Y 109.744,Z 295.93,A -85,B 0,C 180,E1 -27757.285,E2 -27757.285} C_VEL
LIN {X 0,Y 107.449,Z 308.881,A -85,B 0,C 180,E1 -27758.472,E2 -27758.472} C_VEL
LIN {X 0,Y 104.367,Z 321.942,A -85,B 0,C 180,E1 -27760.374,E2 -27760.374} C_VEL
LIN {X 0,Y 100.572,Z 333.84,A -85,B 0,C 180,E1 -27762.794,E2 -27762.794} C_VEL
LIN {X 0,Y 96.309,Z 345.35,A -85,B 0,C 180,E1 -27766.107,E2 -27766.107} C_VEL
LIN {X 0,Y 91.762,Z 355.971,A -85,B 0,C 180,E1 -27770.245,E2 -27770.245} C_VEL
LIN {X 0,Y 87.054,Z 365.912,A -85,B 0,C 180,E1 -27775.584,E2 -27775.584} C_VEL
LIN {X 0,Y 82.808,Z 374.844,A -85,B 0,C 180,E1 -27782.169,E2 -27782.169} C_VEL
LIN {X 0,Y 79.6,Z 381.96,A -85,B 0,C 180,E1 -27789.314,E2 -27789.314} C_VEL
LIN {X 0,Y 77.674,Z 387.627,A -85,B 0,C 180,E1 -27796.921,E2 -27796.921} C_VEL
LIN {X 0,Y 76.838,Z 392.04,A -85,B 0,C 180,E1 -27804.747,E2 -27804.747} C_VEL
LIN {X 0,Y 76.836,Z 394.346,A -85,B 0,C 180,E1 -27809.995,E2 -27809.995} C_VEL
LIN {X 0,Y 76.868,Z 396.181,A -85,B 0,C 180,E1 -27815.24,E2 -27815.24} C_VEL
LIN {X 0,Y 77.322,Z 397.588,A -85,B 0,C 180,E1 -27820.468,E2 -27820.468} C_VEL
LIN {X 0,Y 79.829,Z 399.187,A -85,B 0,C 180,E1 -27830.613,E2 -27830.613} C_VEL
LIN {X 0,Y 84.553,Z 399.343,A -85,B 0,C 180,E1 -27839.909,E2 -27839.909} C_VEL
LIN {X 0,Y 91.493,Z 398.011,A -85,B 0,C 180,E1 -27847.91,E2 -27847.91} C_VEL
LIN {X 0,Y 99.977,Z 395.165,A -85,B 0,C 180,E1 -27854.658,E2 -27854.658} C_VEL
LIN {X 0,Y 105.649,Z 392.673,A -85,B 0,C 180,E1 -27858.298,E2 -27858.298} C_VEL
LIN {X 0,Y 114.806,Z 387.84,A -85,B 0,C 180,E1 -27862.725,E2 -27862.725} C_VEL
LIN {X 0,Y 123.014,Z 382.589,A -85,B 0,C 180,E1 -27865.929,E2 -27865.929} C_VEL
LIN {X 0,Y 131.616,Z 376.083,A -85,B 0,C 180,E1 -27868.682,E2 -27868.682} C_VEL
LIN {X 0,Y 140.516,Z 368.124,A -85,B 0,C 180,E1 -27871.069,E2 -27871.069} C_VEL
LIN {X 0,Y 148.135,Z 360.052,A -85,B 0,C 180,E1 -27872.81,E2 -27872.81} C_VEL
LIN {X 0,Y 155.901,Z 350.255,A -85,B 0,C 180,E1 -27874.361,E2 -27874.361} C_VEL
LIN {X 0,Y 163.04,Z 339.301,A -85,B 0,C 180,E1 -27875.582,E2 -27875.582} C_VEL
LIN {X 0,Y 169.098,Z 327.778,A -85,B 0,C 180,E1 -27876.548,E2 -27876.548} C_VEL
LIN {X 0,Y 174.071,Z 315.67,A -85,B 0,C 180,E1 -27877.252,E2 -27877.252} C_VEL
LIN {X 0,Y 177.623,Z 304.109,A -85,B 0,C 180,E1 -27877.748,E2 -27877.748} C_VEL
LIN {X 0,Y 177.6,Z 302.737,A -85,B 0,C 180,E1 -27879.394,E2 -27879.394} C_VEL
LIN {X 0,Y 177.514,Z 302.367,A -85,B 0,C 180,E1 -27883.909,E2 -27883.909} C_VEL
LIN {X 0,Y 177.781,Z 303.04,A -85,B 0,C 180,E1 -27886.278,E2 -27886.278} C_VEL
LIN {X 0,Y 177.77,Z 303.331,A -85,B 0,C 180,E1 -27886.532,E2 -27886.532} C_VEL
LIN {X 0,Y 174.329,Z 314.627,A -85,B 0,C 180,E1 -27887.019,E2 -27887.019} C_VEL
LIN {X 0,Y 172.228,Z 320.157,A -85,B 0,C 180,E1 -27887.108,E2 -27887.108} C_VEL
LIN {X 0,Y 168.006,Z 329.084,A -85,B 0,C 180,E1 -27886.753,E2 -27886.753} C_VEL
LIN {X 0,Y 163.127,Z 337.627,A -85,B 0,C 180,E1 -27886.482,E2 -27886.482} C_VEL
LIN {X 0,Y 159.987,Z 342.545,A -85,B 0,C 180,E1 -27886.732,E2 -27886.732} C_VEL
LIN {X 0,Y 151.698,Z 353.953,A -85,B 0,C 180,E1 -27888.135,E2 -27888.135} C_VEL
LIN {X 0,Y 142.75,Z 363.97,A -85,B 0,C 180,E1 -27889.929,E2 -27889.929} C_VEL
LIN {X 0,Y 134.945,Z 371.258,A -85,B 0,C 180,E1 -27891.674,E2 -27891.674} C_VEL
LIN {X 0,Y 125.372,Z 378.753,A -85,B 0,C 180,E1 -27894.235,E2 -27894.235} C_VEL
LIN {X 0,Y 115.21,Z 385.275,A -85,B 0,C 180,E1 -27897.537,E2 -27897.537} C_VEL
LIN {X 0,Y 105.455,Z 390.291,A -85,B 0,C 180,E1 -27901.653,E2 -27901.653} C_VEL
LIN {X 0,Y 98.78,Z 393.096,A -85,B 0,C 180,E1 -27905.135,E2 -27905.135} C_VEL
LIN {X 0,Y 92.522,Z 395.172,A -85,B 0,C 180,E1 -27909.109,E2 -27909.109} C_VEL
LIN {X 0,Y 86.206,Z 396.743,A -85,B 0,C 180,E1 -27914.155,E2 -27914.155} C_VEL
LIN {X 0,Y 80.228,Z 397.583,A -85,B 0,C 180,E1 -27920.509,E2 -27920.509} C_VEL
LIN {X 0,Y 75.393,Z 397.516,A -85,B 0,C 180,E1 -27927.778,E2 -27927.778} C_VEL
LIN {X 0,Y 71.214,Z 396.16,A -85,B 0,C 180,E1 -27937.871,E2 -27937.871} C_VEL
LIN {X 0,Y 69.17,Z 393.421,A -85,B 0,C 180,E1 -27948.676,E2 -27948.676} C_VEL
LIN {X 0,Y 69.302,Z 389.286,A -85,B 0,C 180,E1 -27959.54,E2 -27959.54} C_VEL
LIN {X 0,Y 70.735,Z 384.708,A -85,B 0,C 180,E1 -27968.131,E2 -27968.131} C_VEL
LIN {X 0,Y 73.4,Z 378.184,A -85,B 0,C 180,E1 -27977.15,E2 -27977.15} C_VEL
LIN {X 0,Y 77.095,Z 370.639,A -85,B 0,C 180,E1 -27984.775,E2 -27984.775} C_VEL
LIN {X 0,Y 81.527,Z 361.912,A -85,B 0,C 180,E1 -27991.241,E2 -27991.241} C_VEL
LIN {X 0,Y 86.369,Z 352.155,A -85,B 0,C 180,E1 -27996.429,E2 -27996.429} C_VEL
LIN {X 0,Y 91.023,Z 341.765,A -85,B 0,C 180,E1 -28000.481,E2 -28000.481} C_VEL
LIN {X 0,Y 95.528,Z 330.019,A -85,B 0,C 180,E1 -28003.838,E2 -28003.838} C_VEL
LIN {X 0,Y 99.535,Z 317.159,A -85,B 0,C 180,E1 -28006.41,E2 -28006.41} C_VEL
LIN {X 0,Y 102.621,Z 304.024,A -85,B 0,C 180,E1 -28008.239,E2 -28008.239} C_VEL
LIN {X 0,Y 104.812,Z 290.598,A -85,B 0,C 180,E1 -28009.366,E2 -28009.366} C_VEL
LIN {X 0,Y 108.182,Z 257.369,A -85,B 0,C 180,E1 -28011.272,E2 -28011.272} C_VEL
LIN {X 0,Y 103.007,Z 245.34,A -85,B 0,C 180,E1 -28015.597,E2 -28015.597} C_VEL
LIN {X 0,Y 97.547,Z 235.226,A -85,B 0,C 180,E1 -28020.645,E2 -28020.645} C_VEL
LIN {X 0,Y 93.912,Z 229.213,A -85,B 0,C 180,E1 -28024.598,E2 -28024.598} C_VEL
LIN {X 0,Y 91.23,Z 225.04,A -85,B 0,C 180,E1 -28027.902,E2 -28027.902} C_VEL
LIN {X 0,Y 89.323,Z 222.101,A -85,B 0,C 180,E1 -28030.56,E2 -28030.56} C_VEL
LIN {X 0,Y 86.857,Z 218.68,A -85,B 0,C 180,E1 -28034.456,E2 -28034.456} C_VEL
LIN {X 0,Y 86.138,Z 217.76,A -85,B 0,C 180,E1 -28035.703,E2 -28035.703} C_VEL
LIN {X 0,Y 83.775,Z 215.009,A -85,B 0,C 180,E1 -28040.431,E2 -28040.431} C_VEL
LIN {X 0,Y 82.789,Z 212.901,A -85,B 0,C 180,E1 -28043.166,E2 -28043.166} C_VEL
LIN {X 0,Y 79.407,Z 209.817,A -85,B 0,C 180,E1 -28057.907,E2 -28057.907} C_VEL
LIN {X 0,Y 79.393,Z 209.284,A -85,B 0,C 180,E1 -28064.602,E2 -28064.602} C_VEL
LIN {X 0,Y 80.144,Z 210.204,A -85,B 0,C 180,E1 -28071.175,E2 -28071.175} C_VEL
LIN {X 0,Y 83.253,Z 212.558,A -85,B 0,C 180,E1 -28081.512,E2 -28081.512} C_VEL
LIN {X 0,Y 84.964,Z 215.887,A -85,B 0,C 180,E1 -28085.676,E2 -28085.676} C_VEL
LIN {X 0,Y 86.867,Z 218.089,A -85,B 0,C 180,E1 -28089.167,E2 -28089.167} C_VEL
LIN {X 0,Y 89.106,Z 221.674,A -85,B 0,C 180,E1 -28092.868,E2 -28092.868} C_VEL
LIN {X 0,Y 92.914,Z 227.582,A -85,B 0,C 180,E1 -28097.984,E2 -28097.984} C_VEL
LIN {X 0,Y 96.722,Z 233.891,A -85,B 0,C 180,E1 -28102.286,E2 -28102.286} C_VEL
LIN {X 0,Y 101.578,Z 243.235,A -85,B 0,C 180,E1 -28107.015,E2 -28107.015} C_VEL
LIN {X 0,Y 104.505,Z 249.951,A -85,B 0,C 180,E1 -28109.632,E2 -28109.632} C_VEL
LIN {X 0,Y 107.951,Z 261.343,A -85,B 0,C 180,E1 -28112.802,E2 -28112.802} C_VEL
LIN {X 0,Y 104.44,Z 295.46,A -85,B 0,C 180,E1 -28114.786,E2 -28114.786} C_VEL
LIN {X 0,Y 102.047,Z 308.529,A -85,B 0,C 180,E1 -28115.974,E2 -28115.974} C_VEL
LIN {X 0,Y 98.96,Z 321.087,A -85,B 0,C 180,E1 -28117.801,E2 -28117.801} C_VEL
LIN {X 0,Y 95.282,Z 332.377,A -85,B 0,C 180,E1 -28120.064,E2 -28120.064} C_VEL
LIN {X 0,Y 90.759,Z 344.163,A -85,B 0,C 180,E1 -28123.445,E2 -28123.445} C_VEL
LIN {X 0,Y 85.975,Z 354.794,A -85,B 0,C 180,E1 -28127.628,E2 -28127.628} C_VEL
LIN {X 0,Y 81.259,Z 364.279,A -85,B 0,C 180,E1 -28132.735,E2 -28132.735} C_VEL
LIN {X 0,Y 76.608,Z 373.48,A -85,B 0,C 180,E1 -28139.691,E2 -28139.691} C_VEL
LIN {X 0,Y 72.984,Z 380.849,A -85,B 0,C 180,E1 -28147.339,E2 -28147.339} C_VEL
LIN {X 0,Y 70.758,Z 386.746,A -85,B 0,C 180,E1 -28155.617,E2 -28155.617} C_VEL
LIN {X 0,Y 69.775,Z 391.329,A -85,B 0,C 180,E1 -28164.213,E2 -28164.213} C_VEL
LIN {X 0,Y 69.747,Z 393.723,A -85,B 0,C 180,E1 -28169.994,E2 -28169.994} C_VEL
LIN {X 0,Y 69.826,Z 395.632,A -85,B 0,C 180,E1 -28175.77,E2 -28175.77} C_VEL
LIN {X 0,Y 70.362,Z 397.129,A -85,B 0,C 180,E1 -28181.517,E2 -28181.517} C_VEL
LIN {X 0,Y 73.2,Z 398.954,A -85,B 0,C 180,E1 -28192.578,E2 -28192.578} C_VEL
LIN {X 0,Y 78.474,Z 399.272,A -85,B 0,C 180,E1 -28202.497,E2 -28202.497} C_VEL
LIN {X 0,Y 85.99,Z 398.166,A -85,B 0,C 180,E1 -28210.825,E2 -28210.825} C_VEL
LIN {X 0,Y 95.061,Z 395.533,A -85,B 0,C 180,E1 -28217.666,E2 -28217.666} C_VEL
LIN {X 0,Y 102.52,Z 392.555,A -85,B 0,C 180,E1 -28222.021,E2 -28222.021} C_VEL
LIN {X 0,Y 110.684,Z 388.589,A -85,B 0,C 180,E1 -28225.626,E2 -28225.626} C_VEL
LIN {X 0,Y 119.218,Z 383.588,A -85,B 0,C 180,E1 -28228.728,E2 -28228.728} C_VEL
LIN {X 0,Y 128.119,Z 377.361,A -85,B 0,C 180,E1 -28231.356,E2 -28231.356} C_VEL
LIN {X 0,Y 137.282,Z 369.677,A -85,B 0,C 180,E1 -28233.615,E2 -28233.615} C_VEL
LIN {X 0,Y 146.668,Z 360.208,A -85,B 0,C 180,E1 -28235.557,E2 -28235.557} C_VEL
LIN {X 0,Y 154.654,Z 350.494,A -85,B 0,C 180,E1 -28236.95,E2 -28236.95} C_VEL
LIN {X 0,Y 161.94,Z 339.691,A -85,B 0,C 180,E1 -28238.062,E2 -28238.062} C_VEL
LIN {X 0,Y 168.489,Z 327.617,A -85,B 0,C 180,E1 -28238.97,E2 -28238.97} C_VEL
LIN {X 0,Y 173.602,Z 315.411,A -85,B 0,C 180,E1 -28239.605,E2 -28239.605} C_VEL
LIN {X 0,Y 175.612,Z 309.378,A -85,B 0,C 180,E1 -28239.892,E2 -28239.892} C_VEL
LIN {X 0,Y 175.615,Z 309.265,A -85,B 0,C 180,E1 -28244.463,E2 -28244.463} C_VEL
LIN {X 0,Y 171.401,Z 320.936,A -85,B 0,C 180,E1 -28245.025,E2 -28245.025} C_VEL
LIN {X 0,Y 165.804,Z 332.709,A -85,B 0,C 180,E1 -28245.824,E2 -28245.824} C_VEL
LIN {X 0,Y 159.987,Z 342.545,A -85,B 0,C 180,E1 -28246.732,E2 -28246.732} C_VEL
LIN {X 0,Y 157.725,Z 345.86,A -85,B 0,C 180,E1 -28246.836,E2 -28246.836} C_VEL
LIN {X 0,Y 149.326,Z 356.194,A -85,B 0,C 180,E1 -28245.948,E2 -28245.948} C_VEL
LIN {X 0,Y 146.663,Z 359.088,A -85,B 0,C 180,E1 -28246.143,E2 -28246.143} C_VEL
LIN {X 0,Y 138.49,Z 367.24,A -85,B 0,C 180,E1 -28247.639,E2 -28247.639} C_VEL
LIN {X 0,Y 128.54,Z 375.468,A -85,B 0,C 180,E1 -28249.765,E2 -28249.765} C_VEL
LIN {X 0,Y 118.161,Z 382.549,A -85,B 0,C 180,E1 -28252.489,E2 -28252.489} C_VEL
LIN {X 0,Y 109.627,Z 387.283,A -85,B 0,C 180,E1 -28255.166,E2 -28255.166} C_VEL
LIN {X 0,Y 98.384,Z 392.259,A -85,B 0,C 180,E1 -28259.828,E2 -28259.828} C_VEL
LIN {X 0,Y 89.791,Z 395.092,A -85,B 0,C 180,E1 -28264.487,E2 -28264.487} C_VEL
LIN {X 0,Y 82.222,Z 396.856,A -85,B 0,C 180,E1 -28269.841,E2 -28269.841} C_VEL
LIN {X 0,Y 73.921,Z 397.753,A -85,B 0,C 180,E1 -28278.079,E2 -28278.079} C_VEL
LIN {X 0,Y 69.498,Z 397.581,A -85,B 0,C 180,E1 -28284.493,E2 -28284.493} C_VEL
LIN {X 0,Y 65.704,Z 396.655,A -85,B 0,C 180,E1 -28292.328,E2 -28292.328} C_VEL
LIN {X 0,Y 62.915,Z 394.69,A -85,B 0,C 180,E1 -28302.082,E2 -28302.082} C_VEL
LIN {X 0,Y 61.889,Z 391.605,A -85,B 0,C 180,E1 -28312.641,E2 -28312.641} C_VEL
LIN {X 0,Y 62.699,Z 387.093,A -85,B 0,C 180,E1 -28323.725,E2 -28323.725} C_VEL
LIN {X 0,Y 64.818,Z 381.691,A -85,B 0,C 180,E1 -28333.328,E2 -28333.328} C_VEL
LIN {X 0,Y 68.263,Z 374.539,A -85,B 0,C 180,E1 -28342.612,E2 -28342.612} C_VEL
LIN {X 0,Y 72.56,Z 366.648,A -85,B 0,C 180,E1 -28350.006,E2 -28350.006} C_VEL
LIN {X 0,Y 77.794,Z 357.007,A -85,B 0,C 180,E1 -28356.431,E2 -28356.431} C_VEL
LIN {X 0,Y 83.232,Z 346.046,A -85,B 0,C 180,E1 -28361.574,E2 -28361.574} C_VEL
LIN {X 0,Y 87.815,Z 335.6,A -85,B 0,C 180,E1 -28365.081,E2 -28365.081} C_VEL
LIN {X 0,Y 92.305,Z 323.303,A -85,B 0,C 180,E1 -28368.022,E2 -28368.022} C_VEL
LIN {X 0,Y 95.794,Z 311.032,A -85,B 0,C 180,E1 -28370.119,E2 -28370.119} C_VEL
LIN {X 0,Y 98.521,Z 298.254,A -85,B 0,C 180,E1 -28371.559,E2 -28371.559} C_VEL
LIN {X 0,Y 100.75,Z 281.332,A -85,B 0,C 180,E1 -28372.646,E2 -28372.646} C_VEL
LIN {X 0,Y 102.94,Z 259.497,A -85,B 0,C 180,E1 -28373.945,E2 -28373.945} C_VEL
LIN {X 0,Y 98.891,Z 249.853,A -85,B 0,C 180,E1 -28377.683,E2 -28377.683} C_VEL
LIN {X 0,Y 93.963,Z 240.157,A -85,B 0,C 180,E1 -28382.841,E2 -28382.841} C_VEL
LIN {X 0,Y 90.742,Z 234.595,A -85,B 0,C 180,E1 -28386.722,E2 -28386.722} C_VEL
LIN {X 0,Y 87.14,Z 228.517,A -85,B 0,C 180,E1 -28391.937,E2 -28391.937} C_VEL
LIN {X 0,Y 84.545,Z 224.671,A -85,B 0,C 180,E1 -28396.477,E2 -28396.477} C_VEL
LIN {X 0,Y 81.887,Z 221.294,A -85,B 0,C 180,E1 -28402.304,E2 -28402.304} C_VEL
LIN {X 0,Y 81.129,Z 219.618,A -85,B 0,C 180,E1 -28404.683,E2 -28404.683} C_VEL
LIN {X 0,Y 78.32,Z 216.723,A -85,B 0,C 180,E1 -28418.967,E2 -28418.967} C_VEL
LIN {X 0,Y 78.354,Z 216.321,A -85,B 0,C 180,E1 -28424.393,E2 -28424.393} C_VEL
LIN {X 0,Y 78.965,Z 217.123,A -85,B 0,C 180,E1 -28430.396,E2 -28430.396} C_VEL
LIN {X 0,Y 81.554,Z 219.24,A -85,B 0,C 180,E1 -28440.002,E2 -28440.002} C_VEL
LIN {X 0,Y 83.386,Z 222.79,A -85,B 0,C 180,E1 -28444.837,E2 -28444.837} C_VEL
LIN {X 0,Y 84.695,Z 224.47,A -85,B 0,C 180,E1 -28447.445,E2 -28447.445} C_VEL
LIN {X 0,Y 87.776,Z 229.621,A -85,B 0,C 180,E1 -28452.858,E2 -28452.858} C_VEL
LIN {X 0,Y 91.367,Z 235.507,A -85,B 0,C 180,E1 -28457.807,E2 -28457.807} C_VEL
LIN {X 0,Y 95.406,Z 243.213,A -85,B 0,C 180,E1 -28462.593,E2 -28462.593} C_VEL
LIN {X 0,Y 99.534,Z 252.242,A -85,B 0,C 180,E1 -28466.821,E2 -28466.821} C_VEL
LIN {X 0,Y 102.661,Z 262.65,A -85,B 0,C 180,E1 -28470.04,E2 -28470.04} C_VEL
LIN {X 0,Y 102.627,Z 264.931,A -85,B 0,C 180,E1 -28470.289,E2 -28470.289} C_VEL
LIN {X 0,Y 99.24,Z 295.64,A -85,B 0,C 180,E1 -28472.059,E2 -28472.059} C_VEL
LIN {X 0,Y 96.685,Z 308.889,A -85,B 0,C 180,E1 -28473.281,E2 -28473.281} C_VEL
LIN {X 0,Y 93.448,Z 321.329,A -85,B 0,C 180,E1 -28475.12,E2 -28475.12} C_VEL
LIN {X 0,Y 89.601,Z 332.543,A -85,B 0,C 180,E1 -28477.417,E2 -28477.417} C_VEL
LIN {X 0,Y 84.828,Z 344.243,A -85,B 0,C 180,E1 -28480.88,E2 -28480.88} C_VEL
LIN {X 0,Y 79.798,Z 354.765,A -85,B 0,C 180,E1 -28485.198,E2 -28485.198} C_VEL
LIN {X 0,Y 74.769,Z 364.261,A -85,B 0,C 180,E1 -28490.613,E2 -28490.613} C_VEL
LIN {X 0,Y 69.778,Z 373.42,A -85,B 0,C 180,E1 -28498.07,E2 -28498.07} C_VEL
LIN {X 0,Y 65.942,Z 380.763,A -85,B 0,C 180,E1 -28506.436,E2 -28506.436} C_VEL
LIN {X 0,Y 63.899,Z 385.729,A -85,B 0,C 180,E1 -28514.033,E2 -28514.033} C_VEL
LIN {X 0,Y 62.733,Z 390.509,A -85,B 0,C 180,E1 -28523.561,E2 -28523.561} C_VEL
LIN {X 0,Y 62.673,Z 393.064,A -85,B 0,C 180,E1 -28529.993,E2 -28529.993} C_VEL
LIN {X 0,Y 62.802,Z 395.076,A -85,B 0,C 180,E1 -28536.418,E2 -28536.418} C_VEL
LIN {X 0,Y 64.71,Z 397.849,A -85,B 0,C 180,E1 -28549.008,E2 -28549.008} C_VEL
LIN {X 0,Y 69.283,Z 399.129,A -85,B 0,C 180,E1 -28560.47,E2 -28560.47} C_VEL
LIN {X 0,Y 76.448,Z 398.915,A -85,B 0,C 180,E1 -28570.047,E2 -28570.047} C_VEL
LIN {X 0,Y 85.436,Z 397.263,A -85,B 0,C 180,E1 -28577.752,E2 -28577.752} C_VEL
LIN {X 0,Y 90.437,Z 395.887,A -85,B 0,C 180,E1 -28580.988,E2 -28580.988} C_VEL
LIN {X 0,Y 98.326,Z 393.074,A -85,B 0,C 180,E1 -28585.271,E2 -28585.271} C_VEL
LIN {X 0,Y 106.869,Z 389.306,A -85,B 0,C 180,E1 -28588.741,E2 -28588.741} C_VEL
LIN {X 0,Y 115.726,Z 384.517,A -85,B 0,C 180,E1 -28591.703,E2 -28591.703} C_VEL
LIN {X 0,Y 124.914,Z 378.545,A -85,B 0,C 180,E1 -28594.175,E2 -28594.175} C_VEL
LIN {X 0,Y 134.335,Z 371.219,A -85,B 0,C 180,E1 -28596.274,E2 -28596.274} C_VEL
LIN {X 0,Y 143.946,Z 362.175,A -85,B 0,C 180,E1 -28598.062,E2 -28598.062} C_VEL
LIN {X 0,Y 152.082,Z 352.926,A -85,B 0,C 180,E1 -28599.346,E2 -28599.346} C_VEL
LIN {X 0,Y 159.505,Z 342.749,A -85,B 0,C 180,E1 -28600.348,E2 -28600.348} C_VEL
LIN {X 0,Y 166.466,Z 330.932,A -85,B 0,C 180,E1 -28601.211,E2 -28601.211} C_VEL
LIN {X 0,Y 172.299,Z 318.096,A -85,B 0,C 180,E1 -28601.849,E2 -28601.849} C_VEL
LIN {X 0,Y 172.816,Z 316.804,A -85,B 0,C 180,E1 -28601.905,E2 -28601.905} C_VEL
LIN {X 0,Y 173.147,Z 315.91,A -85,B 0,C 180,E1 -28602.202,E2 -28602.202} C_VEL
LIN {X 0,Y 172.488,Z 317.59,A -85,B 0,C 180,E1 -28602.457,E2 -28602.457} C_VEL
LIN {X 0,Y 167.044,Z 329.718,A -85,B 0,C 180,E1 -28603.155,E2 -28603.155} C_VEL
LIN {X 0,Y 160.859,Z 340.568,A -85,B 0,C 180,E1 -28603.973,E2 -28603.973} C_VEL
LIN {X 0,Y 154.213,Z 350.085,A -85,B 0,C 180,E1 -28604.922,E2 -28604.922} C_VEL
LIN {X 0,Y 146.663,Z 359.088,A -85,B 0,C 180,E1 -28606.143,E2 -28606.143} C_VEL
LIN {X 0,Y 143.875,Z 361.977,A -85,B 0,C 180,E1 -28606.364,E2 -28606.364} C_VEL
LIN {X 0,Y 138.937,Z 366.588,A -85,B 0,C 180,E1 -28605.99,E2 -28605.99} C_VEL
LIN {X 0,Y 133.835,Z 370.872,A -85,B 0,C 180,E1 -28605.621,E2 -28605.621} C_VEL
LIN {X 0,Y 130.788,Z 373.27,A -85,B 0,C 180,E1 -28605.887,E2 -28605.887} C_VEL
LIN {X 0,Y 120.296,Z 380.599,A -85,B 0,C 180,E1 -28608.112,E2 -28608.112} C_VEL
LIN {X 0,Y 110.388,Z 386.199,A -85,B 0,C 180,E1 -28610.662,E2 -28610.662} C_VEL
LIN {X 0,Y 98.832,Z 391.383,A -85,B 0,C 180,E1 -28614.536,E2 -28614.536} C_VEL
LIN {X 0,Y 91.428,Z 393.953,A -85,B 0,C 180,E1 -28617.719,E2 -28617.719} C_VEL
LIN {X 0,Y 84.354,Z 395.878,A -85,B 0,C 180,E1 -28621.451,E2 -28621.451} C_VEL
LIN {X 0,Y 77.706,Z 397.129,A -85,B 0,C 180,E1 -28625.86,E2 -28625.86} C_VEL
LIN {X 0,Y 71.289,Z 397.826,A -85,B 0,C 180,E1 -28631.369,E2 -28631.369} C_VEL
LIN {X 0,Y 64.926,Z 397.762,A -85,B 0,C 180,E1 -28638.947,E2 -28638.947} C_VEL
LIN {X 0,Y 59.912,Z 396.783,A -85,B 0,C 180,E1 -28647.981,E2 -28647.981} C_VEL
LIN {X 0,Y 55.919,Z 394.267,A -85,B 0,C 180,E1 -28661.066,E2 -28661.066} C_VEL
LIN {X 0,Y 54.832,Z 390.351,A -85,B 0,C 180,E1 -28674.786,E2 -28674.786} C_VEL
LIN {X 0,Y 55.807,Z 386.225,A -85,B 0,C 180,E1 -28685.331,E2 -28685.331} C_VEL
LIN {X 0,Y 58.268,Z 380.542,A -85,B 0,C 180,E1 -28696.049,E2 -28696.049} C_VEL
LIN {X 0,Y 62.203,Z 373.227,A -85,B 0,C 180,E1 -28705.975,E2 -28705.975} C_VEL
LIN {X 0,Y 66.51,Z 365.911,A -85,B 0,C 180,E1 -28713.035,E2 -28713.035} C_VEL
LIN {X 0,Y 71.807,Z 356.734,A -85,B 0,C 180,E1 -28719.351,E2 -28719.351} C_VEL
LIN {X 0,Y 77.404,Z 346.158,A -85,B 0,C 180,E1 -28724.465,E2 -28724.465} C_VEL
LIN {X 0,Y 82.092,Z 336.046,A -85,B 0,C 180,E1 -28727.954,E2 -28727.954} C_VEL
LIN {X 0,Y 86.582,Z 324.523,A -85,B 0,C 180,E1 -28730.806,E2 -28730.806} C_VEL
LIN {X 0,Y 90.277,Z 312.52,A -85,B 0,C 180,E1 -28732.912,E2 -28732.912} C_VEL
LIN {X 0,Y 93.374,Z 298.943,A -85,B 0,C 180,E1 -28734.513,E2 -28734.513} C_VEL
LIN {X 0,Y 95.452,Z 284.781,A -85,B 0,C 180,E1 -28735.441,E2 -28735.441} C_VEL
LIN {X 0,Y 97.929,Z 261.928,A -85,B 0,C 180,E1 -28736.762,E2 -28736.762} C_VEL
LIN {X 0,Y 94.724,Z 253.941,A -85,B 0,C 180,E1 -28740.16,E2 -28740.16} C_VEL
LIN {X 0,Y 90.378,Z 244.888,A -85,B 0,C 180,E1 -28745.325,E2 -28745.325} C_VEL
LIN {X 0,Y 87.429,Z 239.496,A -85,B 0,C 180,E1 -28749.366,E2 -28749.366} C_VEL
LIN {X 0,Y 84.685,Z 234.552,A -85,B 0,C 180,E1 -28753.932,E2 -28753.932} C_VEL
LIN {X 0,Y 82.209,Z 230.731,A -85,B 0,C 180,E1 -28758.794,E2 -28758.794} C_VEL
LIN {X 0,Y 80.036,Z 227.458,A -85,B 0,C 180,E1 -28764.425,E2 -28764.425} C_VEL
LIN {X 0,Y 79.693,Z 226.474,A -85,B 0,C 180,E1 -28765.733,E2 -28765.733} C_VEL
LIN {X 0,Y 77.304,Z 223.792,A -85,B 0,C 180,E1 -28778.678,E2 -28778.678} C_VEL
LIN {X 0,Y 77.318,Z 223.345,A -85,B 0,C 180,E1 -28784.178,E2 -28784.178} C_VEL
LIN {X 0,Y 77.907,Z 224.252,A -85,B 0,C 180,E1 -28790.4,E2 -28790.4} C_VEL
LIN {X 0,Y 79.954,Z 226.039,A -85,B 0,C 180,E1 -28798.586,E2 -28798.586} C_VEL
LIN {X 0,Y 82.049,Z 229.934,A -85,B 0,C 180,E1 -28804.453,E2 -28804.453} C_VEL
LIN {X 0,Y 85.136,Z 235.334,A -85,B 0,C 180,E1 -28810.661,E2 -28810.661} C_VEL
LIN {X 0,Y 88.34,Z 241.054,A -85,B 0,C 180,E1 -28815.707,E2 -28815.707} C_VEL
LIN {X 0,Y 91.891,Z 248.174,A -85,B 0,C 180,E1 -28820.365,E2 -28820.365} C_VEL
LIN {X 0,Y 95.637,Z 256.983,A -85,B 0,C 180,E1 -28824.73,E2 -28824.73} C_VEL
LIN {X 0,Y 97.714,Z 264.717,A -85,B 0,C 180,E1 -28827.219,E2 -28827.219} C_VEL
LIN {X 0,Y 94.41,Z 294.648,A -85,B 0,C 180,E1 -28829.016,E2 -28829.016} C_VEL
LIN {X 0,Y 91.978,Z 307.17,A -85,B 0,C 180,E1 -28830.074,E2 -28830.074} C_VEL
LIN {X 0,Y 88.526,Z 320.209,A -85,B 0,C 180,E1 -28831.946,E2 -28831.946} C_VEL
LIN {X 0,Y 84.146,Z 332.469,A -85,B 0,C 180,E1 -28834.427,E2 -28834.427} C_VEL
LIN {X 0,Y 79.133,Z 344.095,A -85,B 0,C 180,E1 -28837.925,E2 -28837.925} C_VEL
LIN {X 0,Y 73.766,Z 354.673,A -85,B 0,C 180,E1 -28842.4,E2 -28842.4} C_VEL
LIN {X 0,Y 68.407,Z 364.167,A -85,B 0,C 180,E1 -28848.095,E2 -28848.095} C_VEL
LIN {X 0,Y 63.01,Z 373.312,A -85,B 0,C 180,E1 -28856.096,E2 -28856.096} C_VEL
LIN {X 0,Y 58.926,Z 380.66,A -85,B 0,C 180,E1 -28865.319,E2 -28865.319} C_VEL
LIN {X 0,Y 56.446,Z 386.525,A -85,B 0,C 180,E1 -28875.573,E2 -28875.573} C_VEL
LIN {X 0,Y 55.572,Z 391.097,A -85,B 0,C 180,E1 -28886.367,E2 -28886.367} C_VEL
LIN {X 0,Y 55.61,Z 393.465,A -85,B 0,C 180,E1 -28893.615,E2 -28893.615} C_VEL
LIN {X 0,Y 56.526,Z 396.164,A -85,B 0,C 180,E1 -28904.391,E2 -28904.391} C_VEL
LIN {X 0,Y 60.305,Z 398.344,A -85,B 0,C 180,E1 -28917.777,E2 -28917.777} C_VEL
LIN {X 0,Y 66.935,Z 399.095,A -85,B 0,C 180,E1 -28929.04,E2 -28929.04} C_VEL
LIN {X 0,Y 75.793,Z 398.379,A -85,B 0,C 180,E1 -28937.876,E2 -28937.876} C_VEL
LIN {X 0,Y 86.152,Z 396.196,A -85,B 0,C 180,E1 -28944.654,E2 -28944.654} C_VEL
LIN {X 0,Y 94.475,Z 393.574,A -85,B 0,C 180,E1 -28948.803,E2 -28948.803} C_VEL
LIN {X 0,Y 103.38,Z 390.011,A -85,B 0,C 180,E1 -28952.09,E2 -28952.09} C_VEL
LIN {X 0,Y 115.663,Z 383.709,A -85,B 0,C 180,E1 -28955.695,E2 -28955.695} C_VEL
LIN {X 0,Y 126.847,Z 376.422,A -85,B 0,C 180,E1 -28958.12,E2 -28958.12} C_VEL
LIN {X 0,Y 136.581,Z 368.634,A -85,B 0,C 180,E1 -28959.887,E2 -28959.887} C_VEL
LIN {X 0,Y 145.95,Z 359.573,A -85,B 0,C 180,E1 -28961.323,E2 -28961.323} C_VEL
LIN {X 0,Y 151.435,Z 353.308,A -85,B 0,C 180,E1 -28962.029,E2 -28962.029} C_VEL
LIN {X 0,Y 151.832,Z 352.803,A -85,B 0,C 180,E1 -28962.512,E2 -28962.512} C_VEL
LIN {X 0,Y 144.573,Z 360.929,A -85,B 0,C 180,E1 -28963.558,E2 -28963.558} C_VEL
LIN {X 0,Y 135.722,Z 369.242,A -85,B 0,C 180,E1 -28964.993,E2 -28964.993} C_VEL
LIN {X 0,Y 130.788,Z 373.27,A -85,B 0,C 180,E1 -28965.887,E2 -28965.887} C_VEL
LIN {X 0,Y 126.168,Z 376.699,A -85,B 0,C 180,E1 -28966.511,E2 -28966.511} C_VEL
LIN {X 0,Y 117.765,Z 381.951,A -85,B 0,C 180,E1 -28966.856,E2 -28966.856} C_VEL
LIN {X 0,Y 109.029,Z 386.562,A -85,B 0,C 180,E1 -28967.317,E2 -28967.317} C_VEL
LIN {X 0,Y 103.921,Z 388.862,A -85,B 0,C 180,E1 -28968.237,E2 -28968.237} C_VEL
LIN {X 0,Y 92.243,Z 393.246,A -85,B 0,C 180,E1 -28972.046,E2 -28972.046} C_VEL
LIN {X 0,Y 84.617,Z 395.372,A -85,B 0,C 180,E1 -28975.261,E2 -28975.261} C_VEL
LIN {X 0,Y 75.813,Z 397.112,A -85,B 0,C 180,E1 -28979.998,E2 -28979.998} C_VEL
LIN {X 0,Y 67.64,Z 397.951,A -85,B 0,C 180,E1 -28985.961,E2 -28985.961} C_VEL
LIN {X 0,Y 58.495,Z 397.664,A -85,B 0,C 180,E1 -28996.047,E2 -28996.047} C_VEL
LIN {X 0,Y 53.89,Z 396.731,A -85,B 0,C 180,E1 -29004.112,E2 -29004.112} C_VEL
LIN {X 0,Y 49.16,Z 394.02,A -85,B 0,C 180,E1 -29018.655,E2 -29018.655} C_VEL
LIN {X 0,Y 47.742,Z 390.074,A -85,B 0,C 180,E1 -29033.937,E2 -29033.937} C_VEL
LIN {X 0,Y 48.497,Z 386.549,A -85,B 0,C 180,E1 -29044.241,E2 -29044.241} C_VEL
LIN {X 0,Y 50.77,Z 381.402,A -85,B 0,C 180,E1 -29055.682,E2 -29055.682} C_VEL
LIN {X 0,Y 54.498,Z 374.772,A -85,B 0,C 180,E1 -29066.315,E2 -29066.315} C_VEL
LIN {X 0,Y 59.545,Z 366.888,A -85,B 0,C 180,E1 -29075.086,E2 -29075.086} C_VEL
LIN {X 0,Y 64.485,Z 358.999,A -85,B 0,C 180,E1 -29081.235,E2 -29081.235} C_VEL
LIN {X 0,Y 70.375,Z 348.924,A -85,B 0,C 180,E1 -29086.691,E2 -29086.691} C_VEL
LIN {X 0,Y 76.144,Z 337.549,A -85,B 0,C 180,E1 -29090.896,E2 -29090.896} C_VEL
LIN {X 0,Y 81.141,Z 325.68,A -85,B 0,C 180,E1 -29093.959,E2 -29093.959} C_VEL
LIN {X 0,Y 85.182,Z 313.398,A -85,B 0,C 180,E1 -29096.142,E2 -29096.142} C_VEL
LIN {X 0,Y 88.562,Z 299.409,A -85,B 0,C 180,E1 -29097.793,E2 -29097.793} C_VEL
LIN {X 0,Y 90.806,Z 284.715,A -85,B 0,C 180,E1 -29098.743,E2 -29098.743} C_VEL
LIN {X 0,Y 93.116,Z 264.198,A -85,B 0,C 180,E1 -29099.93,E2 -29099.93} C_VEL
LIN {X 0,Y 90.776,Z 258.117,A -85,B 0,C 180,E1 -29102.822,E2 -29102.822} C_VEL
LIN {X 0,Y 87.1,Z 249.928,A -85,B 0,C 180,E1 -29107.756,E2 -29107.756} C_VEL
LIN {X 0,Y 83.78,Z 243.257,A -85,B 0,C 180,E1 -29113.207,E2 -29113.207} C_VEL
LIN {X 0,Y 81.967,Z 240.079,A -85,B 0,C 180,E1 -29116.694,E2 -29116.694} C_VEL
LIN {X 0,Y 80.209,Z 237.051,A -85,B 0,C 180,E1 -29120.707,E2 -29120.707} C_VEL
LIN {X 0,Y 78.352,Z 233.788,A -85,B 0,C 180,E1 -29126.409,E2 -29126.409} C_VEL
LIN {X 0,Y 77.933,Z 233.101,A -85,B 0,C 180,E1 -29128.029,E2 -29128.029} C_VEL
LIN {X 0,Y 76.233,Z 230.725,A -85,B 0,C 180,E1 -29139.777,E2 -29139.777} C_VEL
LIN {X 0,Y 76.394,Z 230.511,A -85,B 0,C 180,E1 -29146.163,E2 -29146.163} C_VEL
LIN {X 0,Y 78.411,Z 232.802,A -85,B 0,C 180,E1 -29157.112,E2 -29157.112} C_VEL
LIN {X 0,Y 80.722,Z 237.433,A -85,B 0,C 180,E1 -29164.174,E2 -29164.174} C_VEL
LIN {X 0,Y 83.222,Z 242.226,A -85,B 0,C 180,E1 -29169.524,E2 -29169.524} C_VEL
LIN {X 0,Y 86.181,Z 248.208,A -85,B 0,C 180,E1 -29174.659,E2 -29174.659} C_VEL
LIN {X 0,Y 88.723,Z 253.829,A -85,B 0,C 180,E1 -29178.356,E2 -29178.356} C_VEL
LIN {X 0,Y 91.628,Z 261.11,A -85,B 0,C 180,E1 -29182.165,E2 -29182.165} C_VEL
LIN {X 0,Y 92.961,Z 266.618,A -85,B 0,C 180,E1 -29184.068,E2 -29184.068} C_VEL
LIN {X 0,Y 89.657,Z 294.844,A -85,B 0,C 180,E1 -29185.729,E2 -29185.729} C_VEL
LIN {X 0,Y 86.937,Z 308.043,A -85,B 0,C 180,E1 -29186.856,E2 -29186.856} C_VEL
LIN {X 0,Y 83.194,Z 321.245,A -85,B 0,C 180,E1 -29188.774,E2 -29188.774} C_VEL
LIN {X 0,Y 78.943,Z 332.382,A -85,B 0,C 180,E1 -29191.024,E2 -29191.024} C_VEL
LIN {X 0,Y 73.61,Z 344.067,A -85,B 0,C 180,E1 -29194.56,E2 -29194.56} C_VEL
LIN {X 0,Y 67.928,Z 354.574,A -85,B 0,C 180,E1 -29199.099,E2 -29199.099} C_VEL
LIN {X 0,Y 62.195,Z 364.069,A -85,B 0,C 180,E1 -29205.061,E2 -29205.061} C_VEL
LIN {X 0,Y 56.357,Z 373.21,A -85,B 0,C 180,E1 -29213.668,E2 -29213.668} C_VEL
LIN {X 0,Y 51.916,Z 380.532,A -85,B 0,C 180,E1 -29223.89,E2 -29223.89} C_VEL
LIN {X 0,Y 49.604,Z 385.479,A -85,B 0,C 180,E1 -29233.53,E2 -29233.53} C_VEL
LIN {X 0,Y 48.52,Z 390.239,A -85,B 0,C 180,E1 -29245.838,E2 -29245.838} C_VEL
LIN {X 0,Y 48.58,Z 392.759,A -85,B 0,C 180,E1 -29254.139,E2 -29254.139} C_VEL
LIN {X 0,Y 49.697,Z 395.598,A -85,B 0,C 180,E1 -29266.42,E2 -29266.42} C_VEL
LIN {X 0,Y 51.499,Z 397.01,A -85,B 0,C 180,E1 -29274.158,E2 -29274.158} C_VEL
LIN {X 0,Y 57.462,Z 398.651,A -85,B 0,C 180,E1 -29287.691,E2 -29287.691} C_VEL
LIN {X 0,Y 66.204,Z 398.875,A -85,B 0,C 180,E1 -29297.986,E2 -29297.986} C_VEL
LIN {X 0,Y 76.621,Z 397.678,A -85,B 0,C 180,E1 -29305.63,E2 -29305.63} C_VEL
LIN {X 0,Y 88.012,Z 394.964,A -85,B 0,C 180,E1 -29311.436,E2 -29311.436} C_VEL
LIN {X 0,Y 100.272,Z 390.72,A -85,B 0,C 180,E1 -29315.654,E2 -29315.654} C_VEL
LIN {X 0,Y 109.764,Z 386.382,A -85,B 0,C 180,E1 -29318.176,E2 -29318.176} C_VEL
LIN {X 0,Y 119.478,Z 380.945,A -85,B 0,C 180,E1 -29320.234,E2 -29320.234} C_VEL
LIN {X 0,Y 129.366,Z 374.225,A -85,B 0,C 180,E1 -29321.924,E2 -29321.924} C_VEL
LIN {X 0,Y 130.525,Z 373.312,A -85,B 0,C 180,E1 -29322.646,E2 -29322.646} C_VEL
LIN {X 0,Y 120.349,Z 380.313,A -85,B 0,C 180,E1 -29324.467,E2 -29324.467} C_VEL
LIN {X 0,Y 108.117,Z 386.959,A -85,B 0,C 180,E1 -29327.155,E2 -29327.155} C_VEL
LIN {X 0,Y 103.921,Z 388.862,A -85,B 0,C 180,E1 -29328.237,E2 -29328.237} C_VEL
LIN {X 0,Y 98.739,Z 390.996,A -85,B 0,C 180,E1 -29329.317,E2 -29329.317} C_VEL
LIN {X 0,Y 89.455,Z 393.955,A -85,B 0,C 180,E1 -29330.47,E2 -29330.47} C_VEL
LIN {X 0,Y 81.915,Z 395.783,A -85,B 0,C 180,E1 -29331.583,E2 -29331.583} C_VEL
LIN {X 0,Y 76.506,Z 396.797,A -85,B 0,C 180,E1 -29333.125,E2 -29333.125} C_VEL
LIN {X 0,Y 74.823,Z 397.043,A -85,B 0,C 180,E1 -29333.866,E2 -29333.866} C_VEL
LIN {X 0,Y 64.638,Z 398.077,A -85,B 0,C 180,E1 -29339.997,E2 -29339.997} C_VEL
LIN {X 0,Y 56.596,Z 398.002,A -85,B 0,C 180,E1 -29347.13,E2 -29347.13} C_VEL
LIN {X 0,Y 49.696,Z 397.02,A -85,B 0,C 180,E1 -29356.426,E2 -29356.426} C_VEL
LIN {X 0,Y 44.404,Z 395.118,A -85,B 0,C 180,E1 -29368.343,E2 -29368.343} C_VEL
LIN {X 0,Y 40.925,Z 391.336,A -85,B 0,C 180,E1 -29386.628,E2 -29386.628} C_VEL
LIN {X 0,Y 41.452,Z 386.102,A -85,B 0,C 180,E1 -29405.051,E2 -29405.051} C_VEL
LIN {X 0,Y 44.111,Z 380.671,A -85,B 0,C 180,E1 -29418.555,E2 -29418.555} C_VEL
LIN {X 0,Y 48.263,Z 374.092,A -85,B 0,C 180,E1 -29430.009,E2 -29430.009} C_VEL
LIN {X 0,Y 53.906,Z 366.028,A -85,B 0,C 180,E1 -29439.387,E2 -29439.387} C_VEL
LIN {X 0,Y 59.95,Z 357.038,A -85,B 0,C 180,E1 -29446.26,E2 -29446.26} C_VEL
LIN {X 0,Y 66.393,Z 346.407,A -85,B 0,C 180,E1 -29451.665,E2 -29451.665} C_VEL
LIN {X 0,Y 71.91,Z 335.822,A -85,B 0,C 180,E1 -29455.32,E2 -29455.32} C_VEL
LIN {X 0,Y 76.694,Z 324.767,A -85,B 0,C 180,E1 -29457.958,E2 -29457.958} C_VEL
LIN {X 0,Y 80.927,Z 312.243,A -85,B 0,C 180,E1 -29460.053,E2 -29460.053} C_VEL
LIN {X 0,Y 84.251,Z 298.74,A -85,B 0,C 180,E1 -29461.537,E2 -29461.537} C_VEL
LIN {X 0,Y 86.603,Z 283.615,A -85,B 0,C 180,E1 -29462.425,E2 -29462.425} C_VEL
LIN {X 0,Y 88.634,Z 266.687,A -85,B 0,C 180,E1 -29463.353,E2 -29463.353} C_VEL
LIN {X 0,Y 86.375,Z 260.757,A -85,B 0,C 180,E1 -29466.544,E2 -29466.544} C_VEL
LIN {X 0,Y 83.391,Z 253.585,A -85,B 0,C 180,E1 -29471.431,E2 -29471.431} C_VEL
LIN {X 0,Y 80.275,Z 246.966,A -85,B 0,C 180,E1 -29477.682,E2 -29477.682} C_VEL
LIN {X 0,Y 78.338,Z 243.472,A -85,B 0,C 180,E1 -29482.597,E2 -29482.597} C_VEL
LIN {X 0,Y 76.646,Z 240.013,A -85,B 0,C 180,E1 -29488.839,E2 -29488.839} C_VEL
LIN {X 0,Y 75.214,Z 237.841,A -85,B 0,C 180,E1 -29499.145,E2 -29499.145} C_VEL
LIN {X 0,Y 75.231,Z 237.442,A -85,B 0,C 180,E1 -29503.727,E2 -29503.727} C_VEL
LIN {X 0,Y 75.649,Z 238.167,A -85,B 0,C 180,E1 -29509.294,E2 -29509.294} C_VEL
LIN {X 0,Y 76.996,Z 239.693,A -85,B 0,C 180,E1 -29515.905,E2 -29515.905} C_VEL
LIN {X 0,Y 78.831,Z 243.856,A -85,B 0,C 180,E1 -29522.394,E2 -29522.394} C_VEL
LIN {X 0,Y 81.081,Z 248.58,A -85,B 0,C 180,E1 -29527.819,E2 -29527.819} C_VEL
LIN {X 0,Y 84.044,Z 255.263,A -85,B 0,C 180,E1 -29533.524,E2 -29533.524} C_VEL
LIN {X 0,Y 87.36,Z 264.004,A -85,B 0,C 180,E1 -29538.774,E2 -29538.774} C_VEL
LIN {X 0,Y 88.506,Z 268.334,A -85,B 0,C 180,E1 -29540.558,E2 -29540.558} C_VEL
LIN {X 0,Y 85.34,Z 294.32,A -85,B 0,C 180,E1 -29542.062,E2 -29542.062} C_VEL
LIN {X 0,Y 82.606,Z 307.291,A -85,B 0,C 180,E1 -29543.077,E2 -29543.077} C_VEL
LIN {X 0,Y 78.884,Z 319.997,A -85,B 0,C 180,E1 -29544.809,E2 -29544.809} C_VEL
LIN {X 0,Y 74.068,Z 332.22,A -85,B 0,C 180,E1 -29547.172,E2 -29547.172} C_VEL
LIN {X 0,Y 68.417,Z 343.887,A -85,B 0,C 180,E1 -29550.644,E2 -29550.644} C_VEL
LIN {X 0,Y 62.272,Z 354.532,A -85,B 0,C 180,E1 -29555.283,E2 -29555.283} C_VEL
LIN {X 0,Y 56.195,Z 363.87,A -85,B 0,C 180,E1 -29561.366,E2 -29561.366} C_VEL
LIN {X 0,Y 49.841,Z 373.008,A -85,B 0,C 180,E1 -29570.605,E2 -29570.605} C_VEL
LIN {X 0,Y 44.962,Z 380.34,A -85,B 0,C 180,E1 -29582.025,E2 -29582.025} C_VEL
LIN {X 0,Y 42.143,Z 386.203,A -85,B 0,C 180,E1 -29595.504,E2 -29595.504} C_VEL
LIN {X 0,Y 41.491,Z 390.768,A -85,B 0,C 180,E1 -29609.99,E2 -29609.99} C_VEL
LIN {X 0,Y 41.788,Z 393.115,A -85,B 0,C 180,E1 -29619.672,E2 -29619.672} C_VEL
LIN {X 0,Y 42.957,Z 395.008,A -85,B 0,C 180,E1 -29629.089,E2 -29629.089} C_VEL
LIN {X 0,Y 48.189,Z 397.624,A -85,B 0,C 180,E1 -29645.676,E2 -29645.676} C_VEL
LIN {X 0,Y 52.012,Z 398.389,A -85,B 0,C 180,E1 -29652.489,E2 -29652.489} C_VEL
LIN {X 0,Y 61.663,Z 398.81,A -85,B 0,C 180,E1 -29662.91,E2 -29662.91} C_VEL
LIN {X 0,Y 72.853,Z 397.812,A -85,B 0,C 180,E1 -29670.238,E2 -29670.238} C_VEL
LIN {X 0,Y 84.851,Z 395.397,A -85,B 0,C 180,E1 -29675.644,E2 -29675.644} C_VEL
LIN {X 0,Y 94.343,Z 392.545,A -85,B 0,C 180,E1 -29678.605,E2 -29678.605} C_VEL
LIN {X 0,Y 104.06,Z 388.75,A -85,B 0,C 180,E1 -29680.988,E2 -29680.988} C_VEL
LIN {X 0,Y 110.63,Z 385.68,A -85,B 0,C 180,E1 -29682.33,E2 -29682.33} C_VEL
LIN {X 0,Y 110.42,Z 385.777,A -85,B 0,C 180,E1 -29682.677,E2 -29682.677} C_VEL
LIN {X 0,Y 98.028,Z 391.062,A -85,B 0,C 180,E1 -29685.414,E2 -29685.414} C_VEL
LIN {X 0,Y 85.852,Z 394.845,A -85,B 0,C 180,E1 -29689.184,E2 -29689.184} C_VEL
LIN {X 0,Y 74.823,Z 397.043,A -85,B 0,C 180,E1 -29693.866,E2 -29693.866} C_VEL
LIN {X 0,Y 69.615,Z 397.722,A -85,B 0,C 180,E1 -29696.026,E2 -29696.026} C_VEL
LIN {X 0,Y 60.306,Z 398.203,A -85,B 0,C 180,E1 -29699.03,E2 -29699.03} C_VEL
LIN {X 0,Y 51.237,Z 397.895,A -85,B 0,C 180,E1 -29703.149,E2 -29703.149} C_VEL
LIN {X 0,Y 46.625,Z 397.302,A -85,B 0,C 180,E1 -29707.432,E2 -29707.432} C_VEL
LIN {X 0,Y 38.264,Z 394.856,A -85,B 0,C 180,E1 -29723.344,E2 -29723.344} C_VEL
LIN {X 0,Y 34.013,Z 390.942,A -85,B 0,C 180,E1 -29744.108,E2 -29744.108} C_VEL
LIN {X 0,Y 34.373,Z 385.72,A -85,B 0,C 180,E1 -29765.876,E2 -29765.876} C_VEL
LIN {X 0,Y 37.445,Z 380.153,A -85,B 0,C 180,E1 -29781.919,E2 -29781.919} C_VEL
LIN {X 0,Y 42.318,Z 373.341,A -85,B 0,C 180,E1 -29794.873,E2 -29794.873} C_VEL
LIN {X 0,Y 48.643,Z 365.097,A -85,B 0,C 180,E1 -29804.654,E2 -29804.654} C_VEL
LIN {X 0,Y 55.976,Z 354.906,A -85,B 0,C 180,E1 -29812.135,E2 -29812.135} C_VEL
LIN {X 0,Y 62.351,Z 344.831,A -85,B 0,C 180,E1 -29816.807,E2 -29816.807} C_VEL
LIN {X 0,Y 68.14,Z 333.95,A -85,B 0,C 180,E1 -29820.193,E2 -29820.193} C_VEL
LIN {X 0,Y 73.696,Z 321.131,A -85,B 0,C 180,E1 -29822.852,E2 -29822.852} C_VEL
LIN {X 0,Y 77.753,Z 308.5,A -85,B 0,C 180,E1 -29824.644,E2 -29824.644} C_VEL
LIN {X 0,Y 80.986,Z 294.431,A -85,B 0,C 180,E1 -29825.826,E2 -29825.826} C_VEL
LIN {X 0,Y 84.387,Z 269.075,A -85,B 0,C 180,E1 -29827.126,E2 -29827.126} C_VEL
LIN {X 0,Y 81.221,Z 260.454,A -85,B 0,C 180,E1 -29832.858,E2 -29832.858} C_VEL
LIN {X 0,Y 78.868,Z 254.745,A -85,B 0,C 180,E1 -29837.984,E2 -29837.984} C_VEL
LIN {X 0,Y 76.833,Z 250.256,A -85,B 0,C 180,E1 -29843.716,E2 -29843.716} C_VEL
LIN {X 0,Y 75.229,Z 246.813,A -85,B 0,C 180,E1 -29850.28,E2 -29850.28} C_VEL
LIN {X 0,Y 74.154,Z 244.734,A -85,B 0,C 180,E1 -29860.563,E2 -29860.563} C_VEL
LIN {X 0,Y 74.291,Z 244.566,A -85,B 0,C 180,E1 -29865.763,E2 -29865.763} C_VEL
LIN {X 0,Y 75.548,Z 246.468,A -85,B 0,C 180,E1 -29874.456,E2 -29874.456} C_VEL
LIN {X 0,Y 76.983,Z 250.201,A -85,B 0,C 180,E1 -29880.411,E2 -29880.411} C_VEL
LIN {X 0,Y 79.172,Z 255.432,A -85,B 0,C 180,E1 -29886.493,E2 -29886.493} C_VEL
LIN {X 0,Y 81.672,Z 261.966,A -85,B 0,C 180,E1 -29891.895,E2 -29891.895} C_VEL
LIN {X 0,Y 84.128,Z 269.408,A -85,B 0,C 180,E1 -29896.416,E2 -29896.416} C_VEL
LIN {X 0,Y 84.337,Z 270.457,A -85,B 0,C 180,E1 -29896.84,E2 -29896.84} C_VEL
LIN {X 0,Y 80.899,Z 296.132,A -85,B 0,C 180,E1 -29898.194,E2 -29898.194} C_VEL
LIN {X 0,Y 77.729,Z 309.71,A -85,B 0,C 180,E1 -29899.29,E2 -29899.29} C_VEL
LIN {X 0,Y 73.844,Z 321.805,A -85,B 0,C 180,E1 -29900.937,E2 -29900.937} C_VEL
LIN {X 0,Y 68.819,Z 333.498,A -85,B 0,C 180,E1 -29903.19,E2 -29903.19} C_VEL
LIN {X 0,Y 62.876,Z 344.892,A -85,B 0,C 180,E1 -29906.581,E2 -29906.581} C_VEL
LIN {X 0,Y 56.447,Z 355.186,A -85,B 0,C 180,E1 -29911.119,E2 -29911.119} C_VEL
LIN {X 0,Y 50.496,Z 363.647,A -85,B 0,C 180,E1 -29916.831,E2 -29916.831} C_VEL
LIN {X 0,Y 43.501,Z 372.801,A -85,B 0,C 180,E1 -29926.623,E2 -29926.623} C_VEL
LIN {X 0,Y 38.087,Z 380.151,A -85,B 0,C 180,E1 -29939.494,E2 -29939.494} C_VEL
LIN {X 0,Y 35.317,Z 385.118,A -85,B 0,C 180,E1 -29952.621,E2 -29952.621} C_VEL
LIN {X 0,Y 34.432,Z 389.881,A -85,B 0,C 180,E1 -29969.988,E2 -29969.988} C_VEL
LIN {X 0,Y 35.422,Z 393.403,A -85,B 0,C 180,E1 -29987.301,E2 -29987.301} C_VEL
LIN {X 0,Y 39.004,Z 395.971,A -85,B 0,C 180,E1 -30002.709,E2 -30002.709} C_VEL
LIN {X 0,Y 47.013,Z 398.048,A -85,B 0,C 180,E1 -30018.355,E2 -30018.355} C_VEL
LIN {X 0,Y 57.649,Z 398.731,A -85,B 0,C 180,E1 -30028.565,E2 -30028.565} C_VEL
LIN {X 0,Y 69.607,Z 397.947,A -85,B 0,C 180,E1 -30035.311,E2 -30035.311} C_VEL
LIN {X 0,Y 82.184,Z 395.745,A -85,B 0,C 180,E1 -30040.146,E2 -30040.146} C_VEL
LIN {X 0,Y 88.702,Z 394.089,A -85,B 0,C 180,E1 -30041.931,E2 -30041.931} C_VEL
LIN {X 0,Y 89.72,Z 393.787,A -85,B 0,C 180,E1 -30042.919,E2 -30042.919} C_VEL
LIN {X 0,Y 79.719,Z 396.162,A -85,B 0,C 180,E1 -30045.848,E2 -30045.848} C_VEL
LIN {X 0,Y 71.236,Z 397.477,A -85,B 0,C 180,E1 -30049.085,E2 -30049.085} C_VEL
LIN {X 0,Y 62.449,Z 398.203,A -85,B 0,C 180,E1 -30053.535,E2 -30053.535} C_VEL
LIN {X 0,Y 53.516,Z 398.119,A -85,B 0,C 180,E1 -30059.997,E2 -30059.997} C_VEL
LIN {X 0,Y 46.625,Z 397.302,A -85,B 0,C 180,E1 -30067.432,E2 -30067.432} C_VEL
LIN {X 0,Y 42.349,Z 396.489,A -85,B 0,C 180,E1 -30072.569,E2 -30072.569} C_VEL
LIN {X 0,Y 34.819,Z 394.434,A -85,B 0,C 180,E1 -30081.68,E2 -30081.68} C_VEL
LIN {X 0,Y 29.568,Z 392.237,A -85,B 0,C 180,E1 -30091.684,E2 -30091.684} C_VEL
LIN {X 0,Y 27.112,Z 390.278,A -85,B 0,C 180,E1 -30101.951,E2 -30101.951} C_VEL
LIN {X 0,Y 26.753,Z 389.565,A -85,B 0,C 180,E1 -30105.851,E2 -30105.851} C_VEL
LIN {X 0,Y 27.825,Z 384.155,A -85,B 0,C 180,E1 -30131.612,E2 -30131.612} C_VEL
LIN {X 0,Y 31.096,Z 379.357,A -85,B 0,C 180,E1 -30147.133,E2 -30147.133} C_VEL
LIN {X 0,Y 36.697,Z 372.57,A -85,B 0,C 180,E1 -30161.053,E2 -30161.053} C_VEL
LIN {X 0,Y 44.395,Z 363.478,A -85,B 0,C 180,E1 -30171.707,E2 -30171.707} C_VEL
LIN {X 0,Y 51.934,Z 353.676,A -85,B 0,C 180,E1 -30178.28,E2 -30178.28} C_VEL
LIN {X 0,Y 58.705,Z 343.385,A -85,B 0,C 180,E1 -30182.543,E2 -30182.543} C_VEL
LIN {X 0,Y 64.908,Z 332.066,A -85,B 0,C 180,E1 -30185.597,E2 -30185.597} C_VEL
LIN {X 0,Y 70.13,Z 320.158,A -85,B 0,C 180,E1 -30187.718,E2 -30187.718} C_VEL
LIN {X 0,Y 74.516,Z 306.581,A -85,B 0,C 180,E1 -30189.376,E2 -30189.376} C_VEL
LIN {X 0,Y 77.481,Z 293.607,A -85,B 0,C 180,E1 -30190.269,E2 -30190.269} C_VEL
LIN {X 0,Y 80.476,Z 271.811,A -85,B 0,C 180,E1 -30191.295,E2 -30191.295} C_VEL
LIN {X 0,Y 78.127,Z 264.633,A -85,B 0,C 180,E1 -30196.547,E2 -30196.547} C_VEL
LIN {X 0,Y 75.996,Z 258.861,A -85,B 0,C 180,E1 -30202.531,E2 -30202.531} C_VEL
LIN {X 0,Y 74.817,Z 256.073,A -85,B 0,C 180,E1 -30206.939,E2 -30206.939} C_VEL
LIN {X 0,Y 73.897,Z 253.617,A -85,B 0,C 180,E1 -30211.609,E2 -30211.609} C_VEL
LIN {X 0,Y 73.132,Z 251.62,A -85,B 0,C 180,E1 -30221.803,E2 -30221.803} C_VEL
LIN {X 0,Y 73.277,Z 251.716,A -85,B 0,C 180,E1 -30226.24,E2 -30226.24} C_VEL
LIN {X 0,Y 74.169,Z 253.325,A -85,B 0,C 180,E1 -30233.119,E2 -30233.119} C_VEL
LIN {X 0,Y 75.201,Z 256.44,A -85,B 0,C 180,E1 -30238.203,E2 -30238.203} C_VEL
LIN {X 0,Y 76.838,Z 261.075,A -85,B 0,C 180,E1 -30243.819,E2 -30243.819} C_VEL
LIN {X 0,Y 78.908,Z 267.214,A -85,B 0,C 180,E1 -30249.115,E2 -30249.115} C_VEL
LIN {X 0,Y 80.47,Z 272.607,A -85,B 0,C 180,E1 -30252.649,E2 -30252.649} C_VEL
LIN {X 0,Y 77.287,Z 295.642,A -85,B 0,C 180,E1 -30253.771,E2 -30253.771} C_VEL
LIN {X 0,Y 74.154,Z 308.821,A -85,B 0,C 180,E1 -30254.684,E2 -30254.684} C_VEL
LIN {X 0,Y 69.994,Z 321.424,A -85,B 0,C 180,E1 -30256.21,E2 -30256.21} C_VEL
LIN {X 0,Y 64.744,Z 333.183,A -85,B 0,C 180,E1 -30258.209,E2 -30258.209} C_VEL
LIN {X 0,Y 58.308,Z 344.885,A -85,B 0,C 180,E1 -30261.409,E2 -30261.409} C_VEL
LIN {X 0,Y 51.633,Z 354.929,A -85,B 0,C 180,E1 -30265.593,E2 -30265.593} C_VEL
LIN {X 0,Y 45.182,Z 363.39,A -85,B 0,C 180,E1 -30271.166,E2 -30271.166} C_VEL
LIN {X 0,Y 37.451,Z 372.552,A -85,B 0,C 180,E1 -30281.338,E2 -30281.338} C_VEL
LIN {X 0,Y 31.317,Z 379.9,A -85,B 0,C 180,E1 -30295.857,E2 -30295.857} C_VEL
LIN {X 0,Y 27.818,Z 385.768,A -85,B 0,C 180,E1 -30315.351,E2 -30315.351} C_VEL
LIN {X 0,Y 27.381,Z 388.955,A -85,B 0,C 180,E1 -30329.985,E2 -30329.985} C_VEL
LIN {X 0,Y 28.753,Z 392.68,A -85,B 0,C 180,E1 -30351.492,E2 -30351.492} C_VEL
LIN {X 0,Y 33.256,Z 395.411,A -85,B 0,C 180,E1 -30369.329,E2 -30369.329} C_VEL
LIN {X 0,Y 42.62,Z 397.696,A -85,B 0,C 180,E1 -30385.519,E2 -30385.519} C_VEL
LIN {X 0,Y 54.277,Z 398.572,A -85,B 0,C 180,E1 -30394.991,E2 -30394.991} C_VEL
LIN {X 0,Y 66.949,Z 398.059,A -85,B 0,C 180,E1 -30400.849,E2 -30400.849} C_VEL
LIN {X 0,Y 71.296,Z 397.537,A -85,B 0,C 180,E1 -30402.796,E2 -30402.796} C_VEL
LIN {X 0,Y 57.363,Z 398.398,A -85,B 0,C 180,E1 -30408.52,E2 -30408.52} C_VEL
LIN {X 0,Y 49.509,Z 398.077,A -85,B 0,C 180,E1 -30413.468,E2 -30413.468} C_VEL
LIN {X 0,Y 41.732,Z 397.095,A -85,B 0,C 180,E1 -30420.753,E2 -30420.753} C_VEL
LIN {X 0,Y 34.633,Z 395.327,A -85,B 0,C 180,E1 -30431.703,E2 -30431.703} C_VEL
LIN {X 0,Y 28.879,Z 392.432,A -85,B 0,C 180,E1 -30449.118,E2 -30449.118} C_VEL
LIN {X 0,Y 26.753,Z 389.565,A -85,B 0,C 180,E1 -30465.851,E2 -30465.851} C_VEL
LIN {X 0,Y 25.949,Z 387.321,A -85,B 0,C 180,E1 -30477.62,E2 -30477.62} C_VEL
LIN {X 0,Y 25.21,Z 384.751,A -85,B 0,C 180,E1 -30489.55,E2 -30489.55} C_VEL
LIN {X 0,Y 25.948,Z 378.806,A -85,B 0,C 180,E1 -30513.092,E2 -30513.092} C_VEL
LIN {X 0,Y 28.168,Z 375.446,A -85,B 0,C 180,E1 -30522.548,E2 -30522.548} C_VEL
LIN {X 0,Y 29.212,Z 374.274,A -85,B 0,C 180,E1 -30525.032,E2 -30525.032} C_VEL
LIN {X 0,Y 36.37,Z 366.859,A -85,B 0,C 180,E1 -30535.559,E2 -30535.559} C_VEL
LIN {X 0,Y 44.104,Z 357.982,A -85,B 0,C 180,E1 -30542.545,E2 -30542.545} C_VEL
LIN {X 0,Y 51.312,Z 348.477,A -85,B 0,C 180,E1 -30546.851,E2 -30546.851} C_VEL
LIN {X 0,Y 58.631,Z 336.867,A -85,B 0,C 180,E1 -30550.121,E2 -30550.121} C_VEL
LIN {X 0,Y 64.473,Z 325.282,A -85,B 0,C 180,E1 -30552.209,E2 -30552.209} C_VEL
LIN {X 0,Y 69.179,Z 313.125,A -85,B 0,C 180,E1 -30553.712,E2 -30553.712} C_VEL
LIN {X 0,Y 72.914,Z 299.98,A -85,B 0,C 180,E1 -30554.741,E2 -30554.741} C_VEL
LIN {X 0,Y 75.488,Z 285.677,A -85,B 0,C 180,E1 -30555.311,E2 -30555.311} C_VEL
LIN {X 0,Y 76.948,Z 274.554,A -85,B 0,C 180,E1 -30555.86,E2 -30555.86} C_VEL
LIN {X 0,Y 75.249,Z 268.704,A -85,B 0,C 180,E1 -30560.776,E2 -30560.776} C_VEL
LIN {X 0,Y 73.942,Z 264.467,A -85,B 0,C 180,E1 -30565.71,E2 -30565.71} C_VEL
LIN {X 0,Y 73.029,Z 261.948,A -85,B 0,C 180,E1 -30570.021,E2 -30570.021} C_VEL
LIN {X 0,Y 72.523,Z 260.294,A -85,B 0,C 180,E1 -30573.552,E2 -30573.552} C_VEL
LIN {X 0,Y 72.114,Z 258.547,A -85,B 0,C 180,E1 -30583.003,E2 -30583.003} C_VEL
LIN {X 0,Y 72.335,Z 259.12,A -85,B 0,C 180,E1 -30587.711,E2 -30587.711} C_VEL
LIN {X 0,Y 72.845,Z 260.182,A -85,B 0,C 180,E1 -30591.794,E2 -30591.794} C_VEL
LIN {X 0,Y 73.72,Z 263.353,A -85,B 0,C 180,E1 -30596.864,E2 -30596.864} C_VEL
LIN {X 0,Y 75.103,Z 268.23,A -85,B 0,C 180,E1 -30602.51,E2 -30602.51} C_VEL
LIN {X 0,Y 76.424,Z 273.089,A -85,B 0,C 180,E1 -30606.608,E2 -30606.608} C_VEL
LIN {X 0,Y 77,Z 275.369,A -85,B 0,C 180,E1 -30608.196,E2 -30608.196} C_VEL
LIN {X 0,Y 73.863,Z 296.472,A -85,B 0,C 180,E1 -30609.049,E2 -30609.049} C_VEL
LIN {X 0,Y 70.445,Z 309.996,A -85,B 0,C 180,E1 -30609.846,E2 -30609.846} C_VEL
LIN {X 0,Y 66.251,Z 321.902,A -85,B 0,C 180,E1 -30611.083,E2 -30611.083} C_VEL
LIN {X 0,Y 60.394,Z 334.259,A -85,B 0,C 180,E1 -30612.918,E2 -30612.918} C_VEL
LIN {X 0,Y 54.218,Z 344.836,A -85,B 0,C 180,E1 -30615.468,E2 -30615.468} C_VEL
LIN {X 0,Y 46.605,Z 355.555,A -85,B 0,C 180,E1 -30619.5,E2 -30619.5} C_VEL
LIN {X 0,Y 38.931,Z 364.697,A -85,B 0,C 180,E1 -30625.473,E2 -30625.473} C_VEL
LIN {X 0,Y 30.507,Z 373.592,A -85,B 0,C 180,E1 -30636.241,E2 -30636.241} C_VEL
LIN {X 0,Y 23.814,Z 380.731,A -85,B 0,C 180,E1 -30653.804,E2 -30653.804} C_VEL
LIN {X 0,Y 20.41,Z 386.378,A -85,B 0,C 180,E1 -30680.065,E2 -30680.065} C_VEL
LIN {X 0,Y 20.592,Z 389.398,A -85,B 0,C 180,E1 -30699.804,E2 -30699.804} C_VEL
LIN {X 0,Y 23.953,Z 392.94,A -85,B 0,C 180,E1 -30725.908,E2 -30725.908} C_VEL
LIN {X 0,Y 33.279,Z 396.206,A -85,B 0,C 180,E1 -30747.618,E2 -30747.618} C_VEL
LIN {X 0,Y 39.038,Z 397.298,A -85,B 0,C 180,E1 -30754.152,E2 -30754.152} C_VEL
LIN {X 0,Y 51.672,Z 398.411,A -85,B 0,C 180,E1 -30762.162,E2 -30762.162} C_VEL
LIN {X 0,Y 51.364,Z 398.388,A -85,B 0,C 180,E1 -30763.261,E2 -30763.261} C_VEL
LIN {X 0,Y 40.385,Z 397.316,A -85,B 0,C 180,E1 -30769.973,E2 -30769.973} C_VEL
LIN {X 0,Y 31.313,Z 395.4,A -85,B 0,C 180,E1 -30779.994,E2 -30779.994} C_VEL
LIN {X 0,Y 22.664,Z 391.886,A -85,B 0,C 180,E1 -30801.576,E2 -30801.576} C_VEL
LIN {X 0,Y 19.561,Z 386.679,A -85,B 0,C 180,E1 -30837.921,E2 -30837.921} C_VEL
LIN {X 0,Y 22.546,Z 381.475,A -85,B 0,C 180,E1 -30864.866,E2 -30864.866} C_VEL
LIN {X 0,Y 29.063,Z 374.431,A -85,B 0,C 180,E1 -30884.725,E2 -30884.725} C_VEL
LIN {X 0,Y 29.212,Z 374.274,A -85,B 0,C 180,E1 -30885.032,E2 -30885.032} C_VEL
LIN {X 0,Y 32.167,Z 370.691,A -85,B 0,C 180,E1 -30891.815,E2 -30891.815} C_VEL
LIN {X 0,Y 36.418,Z 364.252,A -85,B 0,C 180,E1 -30902.33,E2 -30902.33} C_VEL
LIN {X 0,Y 41.147,Z 357.309,A -85,B 0,C 180,E1 -30910.164,E2 -30910.164} C_VEL
LIN {X 0,Y 44.528,Z 352.816,A -85,B 0,C 180,E1 -30912.691,E2 -30912.691} C_VEL
LIN {X 0,Y 52.787,Z 341.265,A -85,B 0,C 180,E1 -30915.705,E2 -30915.705} C_VEL
LIN {X 0,Y 59.291,Z 329.807,A -85,B 0,C 180,E1 -30917.55,E2 -30917.55} C_VEL
LIN {X 0,Y 64.84,Z 317.285,A -85,B 0,C 180,E1 -30918.863,E2 -30918.863} C_VEL
LIN {X 0,Y 69.131,Z 304.073,A -85,B 0,C 180,E1 -30919.774,E2 -30919.774} C_VEL
LIN {X 0,Y 72.194,Z 289.634,A -85,B 0,C 180,E1 -30920.284,E2 -30920.284} C_VEL
LIN {X 0,Y 73.884,Z 277.429,A -85,B 0,C 180,E1 -30920.792,E2 -30920.792} C_VEL
LIN {X 0,Y 72.717,Z 272.396,A -85,B 0,C 180,E1 -30925.777,E2 -30925.777} C_VEL
LIN {X 0,Y 71.798,Z 269.068,A -85,B 0,C 180,E1 -30930.7,E2 -30930.7} C_VEL
LIN {X 0,Y 71.27,Z 267.063,A -85,B 0,C 180,E1 -30935.208,E2 -30935.208} C_VEL
LIN {X 0,Y 71.07,Z 265.631,A -85,B 0,C 180,E1 -30942.745,E2 -30942.745} C_VEL
LIN {X 0,Y 71.258,Z 266.168,A -85,B 0,C 180,E1 -30947.373,E2 -30947.373} C_VEL
LIN {X 0,Y 71.552,Z 266.967,A -85,B 0,C 180,E1 -30950.305,E2 -30950.305} C_VEL
LIN {X 0,Y 72.172,Z 269.929,A -85,B 0,C 180,E1 -30954.996,E2 -30954.996} C_VEL
LIN {X 0,Y 73.186,Z 274.573,A -85,B 0,C 180,E1 -30960.262,E2 -30960.262} C_VEL
LIN {X 0,Y 73.904,Z 278.039,A -85,B 0,C 180,E1 -30963.226,E2 -30963.226} C_VEL
LIN {X 0,Y 71.325,Z 295.334,A -85,B 0,C 180,E1 -30963.842,E2 -30963.842} C_VEL
LIN {X 0,Y 67.989,Z 308.65,A -85,B 0,C 180,E1 -30964.385,E2 -30964.385} C_VEL
LIN {X 0,Y 63.533,Z 321.213,A -85,B 0,C 180,E1 -30965.33,E2 -30965.33} C_VEL
LIN {X 0,Y 57.495,Z 333.716,A -85,B 0,C 180,E1 -30966.646,E2 -30966.646} C_VEL
LIN {X 0,Y 50.75,Z 344.849,A -85,B 0,C 180,E1 -30968.679,E2 -30968.679} C_VEL
LIN {X 0,Y 43.062,Z 355.161,A -85,B 0,C 180,E1 -30971.652,E2 -30971.652} C_VEL
LIN {X 0,Y 34.821,Z 364.355,A -85,B 0,C 180,E1 -30976.487,E2 -30976.487} C_VEL
LIN {X 0,Y 25.422,Z 373.282,A -85,B 0,C 180,E1 -30986.007,E2 -30986.007} C_VEL
LIN {X 0,Y 17.408,Z 380.44,A -85,B 0,C 180,E1 -31005.015,E2 -31005.015} C_VEL
LIN {X 0,Y 13.505,Z 385.227,A -85,B 0,C 180,E1 -31034.886,E2 -31034.886} C_VEL
LIN {X 0,Y 13.711,Z 388.429,A -85,B 0,C 180,E1 -31064.819,E2 -31064.819} C_VEL
LIN {X 0,Y 18.701,Z 392.151,A -85,B 0,C 180,E1 -31098.695,E2 -31098.695} C_VEL
LIN {X 0,Y 30.079,Z 395.648,A -85,B 0,C 180,E1 -31119.121,E2 -31119.121} C_VEL
LIN {X 0,Y 32.154,Z 396.052,A -85,B 0,C 180,E1 -31123.976,E2 -31123.976} C_VEL
LIN {X 0,Y 20.152,Z 392.584,A -85,B 0,C 180,E1 -31139.991,E2 -31139.991} C_VEL
LIN {X 0,Y 13.357,Z 388.594,A -85,B 0,C 180,E1 -31171.732,E2 -31171.732} C_VEL
LIN {X 0,Y 14.178,Z 383.102,A -85,B 0,C 180,E1 -31222.376,E2 -31222.376} C_VEL
LIN {X 0,Y 20.967,Z 376.754,A -85,B 0,C 180,E1 -31249.605,E2 -31249.605} C_VEL
LIN {X 0,Y 29.417,Z 369.171,A -85,B 0,C 180,E1 -31262.533,E2 -31262.533} C_VEL
LIN {X 0,Y 38.469,Z 359.921,A -85,B 0,C 180,E1 -31269.762,E2 -31269.762} C_VEL
LIN {X 0,Y 44.528,Z 352.816,A -85,B 0,C 180,E1 -31272.691,E2 -31272.691} C_VEL
LIN {X 0,Y 47.741,Z 348.234,A -85,B 0,C 180,E1 -31274.821,E2 -31274.821} C_VEL
LIN {X 0,Y 52.027,Z 340.303,A -85,B 0,C 180,E1 -31279.531,E2 -31279.531} C_VEL
LIN {X 0,Y 56.016,Z 331.904,A -85,B 0,C 180,E1 -31283.419,E2 -31283.419} C_VEL
LIN {X 0,Y 58.571,Z 326.568,A -85,B 0,C 180,E1 -31284.404,E2 -31284.404} C_VEL
LIN {X 0,Y 63.819,Z 314.067,A -85,B 0,C 180,E1 -31285.089,E2 -31285.089} C_VEL
LIN {X 0,Y 67.971,Z 300.302,A -85,B 0,C 180,E1 -31285.578,E2 -31285.578} C_VEL
LIN {X 0,Y 70.525,Z 286.836,A -85,B 0,C 180,E1 -31285.789,E2 -31285.789} C_VEL
LIN {X 0,Y 71.383,Z 280.616,A -85,B 0,C 180,E1 -31286.055,E2 -31286.055} C_VEL
LIN {X 0,Y 70.644,Z 276.748,A -85,B 0,C 180,E1 -31290.73,E2 -31290.73} C_VEL
LIN {X 0,Y 70.15,Z 273.998,A -85,B 0,C 180,E1 -31295.982,E2 -31295.982} C_VEL
LIN {X 0,Y 70.031,Z 272.695,A -85,B 0,C 180,E1 -31302.481,E2 -31302.481} C_VEL
LIN {X 0,Y 70.196,Z 273.229,A -85,B 0,C 180,E1 -31307.179,E2 -31307.179} C_VEL
LIN {X 0,Y 70.409,Z 274.485,A -85,B 0,C 180,E1 -31310.14,E2 -31310.14} C_VEL
LIN {X 0,Y 71.047,Z 278.746,A -85,B 0,C 180,E1 -31315.704,E2 -31315.704} C_VEL
LIN {X 0,Y 71.403,Z 281.102,A -85,B 0,C 180,E1 -31318.034,E2 -31318.034} C_VEL
LIN {X 0,Y 68.506,Z 298.471,A -85,B 0,C 180,E1 -31318.413,E2 -31318.413} C_VEL
LIN {X 0,Y 65.125,Z 310.814,A -85,B 0,C 180,E1 -31318.712,E2 -31318.712} C_VEL
LIN {X 0,Y 60.628,Z 322.561,A -85,B 0,C 180,E1 -31319.222,E2 -31319.222} C_VEL
LIN {X 0,Y 54.102,Z 335.363,A -85,B 0,C 180,E1 -31320.003,E2 -31320.003} C_VEL
LIN {X 0,Y 47.455,Z 345.73,A -85,B 0,C 180,E1 -31321.133,E2 -31321.133} C_VEL
LIN {X 0,Y 40.46,Z 354.684,A -85,B 0,C 180,E1 -31322.61,E2 -31322.61} C_VEL
LIN {X 0,Y 31.776,Z 363.927,A -85,B 0,C 180,E1 -31325.438,E2 -31325.438} C_VEL
LIN {X 0,Y 21.519,Z 372.876,A -85,B 0,C 180,E1 -31331.446,E2 -31331.446} C_VEL
LIN {X 0,Y 11.857,Z 380.075,A -85,B 0,C 180,E1 -31347.163,E2 -31347.163} C_VEL
LIN {X 0,Y 6.217,Z 385.788,A -85,B 0,C 180,E1 -31409.932,E2 -31409.932} C_VEL
LIN {X 0,Y 9.213,Z 388.786,A -85,B 0,C 180,E1 -31459.644,E2 -31459.644} C_VEL
LIN {X 0,Y 15.011,Z 391.283,A -85,B 0,C 180,E1 -31479.372,E2 -31479.372} C_VEL
LIN {X 0,Y 14.64,Z 391.139,A -85,B 0,C 180,E1 -31483.656,E2 -31483.656} C_VEL
LIN {X 0,Y 7.172,Z 387.682,A -85,B 0,C 180,E1 -31511.782,E2 -31511.782} C_VEL
LIN {X 0,Y 8.418,Z 382.169,A -85,B 0,C 180,E1 -31603.821,E2 -31603.821} C_VEL
LIN {X 0,Y 16.027,Z 376.795,A -85,B 0,C 180,E1 -31626.007,E2 -31626.007} C_VEL
LIN {X 0,Y 26.903,Z 368.091,A -85,B 0,C 180,E1 -31635.945,E2 -31635.945} C_VEL
LIN {X 0,Y 36.626,Z 358.618,A -85,B 0,C 180,E1 -31640.151,E2 -31640.151} C_VEL
LIN {X 0,Y 44.57,Z 349.23,A -85,B 0,C 180,E1 -31642.052,E2 -31642.052} C_VEL
LIN {X 0,Y 52.485,Z 337.709,A -85,B 0,C 180,E1 -31643.471,E2 -31643.471} C_VEL
LIN {X 0,Y 58.571,Z 326.568,A -85,B 0,C 180,E1 -31644.404,E2 -31644.404} C_VEL
LIN {X 0,Y 60.87,Z 321.212,A -85,B 0,C 180,E1 -31645.274,E2 -31645.274} C_VEL
LIN {X 0,Y 63.649,Z 312.226,A -85,B 0,C 180,E1 -31648.156,E2 -31648.156} C_VEL
LIN {X 0,Y 65.851,Z 302.992,A -85,B 0,C 180,E1 -31650.837,E2 -31650.837} C_VEL
LIN {X 0,Y 67.103,Z 297.235,A -85,B 0,C 180,E1 -31651.473,E2 -31651.473} C_VEL
LIN {X 0,Y 69.347,Z 284.13,A -85,B 0,C 180,E1 -31651.624,E2 -31651.624} C_VEL
LIN {X 0,Y 69.049,Z 281.624,A -85,B 0,C 180,E1 -31655.776,E2 -31655.776} C_VEL
LIN {X 0,Y 68.962,Z 280.656,A -85,B 0,C 180,E1 -31658.347,E2 -31658.347} C_VEL
LIN {X 0,Y 68.982,Z 279.84,A -85,B 0,C 180,E1 -31662.206,E2 -31662.206} C_VEL
LIN {X 0,Y 69.072,Z 280.053,A -85,B 0,C 180,E1 -31665.821,E2 -31665.821} C_VEL
LIN {X 0,Y 69.144,Z 281.337,A -85,B 0,C 180,E1 -31668.439,E2 -31668.439} C_VEL
LIN {X 0,Y 69.371,Z 284.372,A -85,B 0,C 180,E1 -31672.413,E2 -31672.413} C_VEL
LIN {X 0,Y 66.68,Z 299.547,A -85,B 0,C 180,E1 -31672.546,E2 -31672.546} C_VEL
LIN {X 0,Y 63.352,Z 311.247,A -85,B 0,C 180,E1 -31672.566,E2 -31672.566} C_VEL
LIN {X 0,Y 58.477,Z 323.546,A -85,B 0,C 180,E1 -31672.583,E2 -31672.583} C_VEL
LIN {X 0,Y 52.093,Z 335.806,A -85,B 0,C 180,E1 -31672.575,E2 -31672.575} C_VEL
LIN {X 0,Y 45.177,Z 346.338,A -85,B 0,C 180,E1 -31672.695,E2 -31672.695} C_VEL
LIN {X 0,Y 37.21,Z 356.129,A -85,B 0,C 180,E1 -31672.646,E2 -31672.646} C_VEL
LIN {X 0,Y 28.349,Z 365.087,A -85,B 0,C 180,E1 -31672.691,E2 -31672.691} C_VEL
LIN {X 0,Y 17.741,Z 373.81,A -85,B 0,C 180,E1 -31672.209,E2 -31672.209} C_VEL
LIN {X 0,Y 7.161,Z 380.77,A -85,B 0,C 180,E1 -31669.24,E2 -31669.24} C_VEL
LIN {X 0,Y 7.681,Z 380.435,A -85,B 0,C 180,E1 -31656.341,E2 -31656.341} C_VEL
LIN {X 0,Y 15.956,Z 375.003,A -85,B 0,C 180,E1 -31651.807,E2 -31651.807} C_VEL
LIN {X 0,Y 25.491,Z 367.519,A -85,B 0,C 180,E1 -31651.164,E2 -31651.164} C_VEL
LIN {X 0,Y 35.094,Z 358.275,A -85,B 0,C 180,E1 -31651.204,E2 -31651.204} C_VEL
LIN {X 0,Y 43.66,Z 348.122,A -85,B 0,C 180,E1 -31651.129,E2 -31651.129} C_VEL
LIN {X 0,Y 51.153,Z 337.163,A -85,B 0,C 180,E1 -31651.163,E2 -31651.163} C_VEL
LIN {X 0,Y 57.686,Z 325.012,A -85,B 0,C 180,E1 -31651.261,E2 -31651.261} C_VEL
LIN {X 0,Y 62.677,Z 312.822,A -85,B 0,C 180,E1 -31651.389,E2 -31651.389} C_VEL
LIN {X 0,Y 66.574,Z 299.644,A -85,B 0,C 180,E1 -31651.49,E2 -31651.49} C_VEL
LIN {X 0,Y 67.103,Z 297.235,A -85,B 0,C 180,E1 -31651.473,E2 -31651.473} C_VEL
LIN {X 0,Y 67.086,Z 296.631,A -85,B 0,C 180,E1 -31652.275,E2 -31652.275} C_VEL
LIN {X 0,Y 66.59,Z 297.357,A -85,B 0,C 180,E1 -31654.447,E2 -31654.447} C_VEL
LIN {X 0,Y 65.538,Z 300.472,A -85,B 0,C 180,E1 -31657.758,E2 -31657.758} C_VEL
LIN {X 0,Y 63.302,Z 308.196,A -85,B 0,C 180,E1 -31662.554,E2 -31662.554} C_VEL
LIN {X 0,Y 61.871,Z 312.74,A -85,B 0,C 180,E1 -31664.62,E2 -31664.62} C_VEL
LIN {X 0,Y 60.165,Z 317.505,A -85,B 0,C 180,E1 -31665.755,E2 -31665.755} C_VEL
LIN {X 0,Y 59.212,Z 319.881,A -85,B 0,C 180,E1 -31665.826,E2 -31665.826} C_VEL
LIN {X 0,Y 53.256,Z 332.307,A -85,B 0,C 180,E1 -31665.018,E2 -31665.018} C_VEL
LIN {X 0,Y 46.612,Z 343.144,A -85,B 0,C 180,E1 -31664.015,E2 -31664.015} C_VEL
LIN {X 0,Y 40.802,Z 351.058,A -85,B 0,C 180,E1 -31662.782,E2 -31662.782} C_VEL
LIN {X 0,Y 40.58,Z 351.325,A -85,B 0,C 180,E1 -31661.082,E2 -31661.082} C_VEL
LIN {X 0,Y 47.804,Z 341.373,A -85,B 0,C 180,E1 -31659.616,E2 -31659.616} C_VEL
LIN {X 0,Y 54.336,Z 330.217,A -85,B 0,C 180,E1 -31658.634,E2 -31658.634} C_VEL
LIN {X 0,Y 60.06,Z 317.703,A -85,B 0,C 180,E1 -31658.023,E2 -31658.023} C_VEL
LIN {X 0,Y 64.229,Z 305.467,A -85,B 0,C 180,E1 -31657.722,E2 -31657.722} C_VEL
LIN {X 0,Y 67.315,Z 291.857,A -85,B 0,C 180,E1 -31657.45,E2 -31657.45} C_VEL
LIN {X 0,Y 67.893,Z 288.32,A -85,B 0,C 180,E1 -31657.512,E2 -31657.512} C_VEL
LIN {X 0,Y 67.894,Z 287.369,A -85,B 0,C 180,E1 -31660.344,E2 -31660.344} C_VEL
LIN {X 0,Y 67.988,Z 286.888,A -85,B 0,C 180,E1 -31664.419,E2 -31664.419} C_VEL
LIN {X 0,Y 67.948,Z 288.079,A -85,B 0,C 180,E1 -31666.547,E2 -31666.547} C_VEL
LIN {X 0,Y 65.498,Z 300.764,A -85,B 0,C 180,E1 -31666.409,E2 -31666.409} C_VEL
LIN {X 0,Y 61.941,Z 312.733,A -85,B 0,C 180,E1 -31666.099,E2 -31666.099} C_VEL
LIN {X 0,Y 59.212,Z 319.881,A -85,B 0,C 180,E1 -31665.826,E2 -31665.826} C_VEL
LIN {X 0,Y 59.063,Z 320.641,A -85,B 0,C 180,E1 -31665.806,E2 -31665.806} C_VEL
LIN {X 0,Y 59.063,Z 600,A -85,B 0,C 180,E1 -31665.806,E2 -31665.806} C_VEL
LIN {X 0,Y 59.063,Z 600,A -85,B 0,C 180,E1 -31665.806,E2 -31665.806}

QRS_NEXT_CUT()

QRS_NEXT()
QRS_HOME()

END
